//--------------------------------------------------------------
// Calculate master max surface speed [m/min]
//--------------------------------------------------------------
masterMaxSpeedMPM := groupMasterMaxSpeedRPM * (PI * upperMasterDiameter) / 1000.0;


//--------------------------------------------------------------
// Determine base speed source (auto/manual) + Recover bump
//--------------------------------------------------------------
IF groupSpeedAutoMan THEN
    baseCmdSpeedMPM := groupAutoSpeedMPM;
ELSE
    baseCmdSpeedMPM := groupManualSpeedMPM;
END_IF;

IF groupRecoverSpeedCmd THEN
    cmdSpeedMPM := baseCmdSpeedMPM + groupRecoverIncrement;
ELSE
    cmdSpeedMPM := baseCmdSpeedMPM;
END_IF;


//--------------------------------------------------------------
// Convert MPM → target RPM for the master
//--------------------------------------------------------------
targetRPM := _Scale(
    X    := cmdSpeedMPM,
    I_LO := 0.0,
    I_HI := masterMaxSpeedMPM,
    O_LO := 0.0,
    O_HI := groupMasterMaxSpeedRPM);


//--------------------------------------------------------------
// Ramp handling
//--------------------------------------------------------------
IF state = 5 OR state = 0 THEN
    // STOPPING — force ramp down to zero speed
    rampTargetRPM := 0.0;

ELSIF state = 10 THEN
    // FAULT — clear ramp immediately to ensure no residual motion
    rampTargetRPM := 0.0;
//    rampReset     := TRUE;

ELSE
    // Normal operation — ramp follows target speed
    rampTargetRPM := targetRPM;
//    rampReset     := FALSE;
END_IF;

// Detect when a new target speed change requires ramping
IF NOT (rampActive AND ABS(rampTargetRPM - baseMasterRefRPM) >= 0.05) OR NOT paperPresenceSensor THEN
   rampActive := TRUE; // Rising edge — ramp request detected
 
END_IF;


IF 	paperPresenceSensor THEN
	//slow	
	instFB_Gen_SRamp.A_UP := MAX(0.0, rampUpRate);
	instFB_Gen_SRamp.A_DN := -MAX(0.0, rampDownRate);

ELSE
	//fast
	instFB_Gen_SRamp.A_UP := MAX(0.0, rampUpRate2);
	instFB_Gen_SRamp.A_DN := -MAX(0.0, rampDownRate2);

END_IF


// Ramp function block execution
instFB_Gen_SRamp(
    X          := rampTargetRPM,
    VU_MAX     := 1000.0,
    VD_MAX     := -1000.0,
    LIMIT_HIGH := groupMasterMaxSpeedRPM,
    RST        := rampReset);


// If ramping, update the baseMasterRefRPM from ramp output
IF rampActive THEN
    baseMasterRefRPM := instFB_Gen_SRamp.Y;

    // Automatically reset ramp flag when the ramp output reaches the target
    IF ABS(instFB_Gen_SRamp.Y - rampTargetRPM) <= 0.05 THEN
        rampActive := FALSE; // Ramp complete
    END_IF;

ELSE
    // No ramping required — direct assignment
    baseMasterRefRPM := rampTargetRPM;
END_IF;


//--------------------------------------------------------------
// Operator offset (TUNE2 control)
//--------------------------------------------------------------
instTUNE2_GroupSpeedDiff(
    SET     := FALSE,
    SU      := groupSpeedDifInc,
    SD      := groupSpeedDifDec,
    RST     := FALSE,
    SS      := speedDifIncPerPulse,
    FS      := speedDifIncPerPulse,
    LIMIT_L := groupSpeedDifLimLow,
    LIMIT_H := groupSpeedDifLimHigh,
    Y       => groupSpeedOffset);

	
speedDif := groupSpeedOffset;
	
groupDeltaRatioAll  := 1.0 + (groupSpeedOffset * 0.01);
upperLowerBiasRatio := 1.0 + ((upperAndLowerSpeedOffset + upperAndLowerSpeedCalibration) * 0.01);


//--------------------------------------------------------------
// Apply offsets + calculate all drive RPM references
//--------------------------------------------------------------
upperMasterRefRPM := baseMasterRefRPM * groupDeltaRatioAll;
upperSlaveRefRPM := upperMasterRefRPM  * upperSlaveRatio;


lowerMasterRefRPM := upperMasterRefRPM * group1ToGroup2MasterRatio;
lowerSlaveRefRPM := lowerMasterRefRPM * lowerSlaveRatio;


//--------------------------------------------------------------
// Convert RPM → MPM (surface speeds)
//--------------------------------------------------------------
upperMasterRefMPM := upperMasterRefRPM * upperMasterDiameter * PI / 1000.0;
upperSlaveRefMPM := (upperSlaveRefRPM * upperSlaveDiameter * PI / 1000.0);


lowerMasterRefMPM := lowerMasterRefRPM * lowerMasterDiameter * PI / 1000.0;
lowerSlaveRefMPM := (lowerSlaveRefRPM * lowerSlaveDiameter * PI / 1000.0);


//--------------------------------------------------------------
// Suggest downstream handoff (group2 master surface speed)
//--------------------------------------------------------------
nextGroupSpeedRefMPM := upperMasterRefMPM;


//====================================================================
// ═══ PRIVATE METHOD — CALCULATE DIAMETER RATIOS ════════════════════
//====================================================================
METHOD PRIVATE _CalculateGearRatios
VAR_INPUT
END_VAR

//──────────────────────────────────────────────────────────────
// Gear Ratios — Group 1 (Reference: Group1 Master)
//──────────────────────────────────────────────────────────────
IF upperMasterDiameter > 0.0 THEN
    group1ToGroup2MasterRatio := upperMasterDiameter / lowerMasterDiameter;
    group1ToGroup1Slave1Ratio := upperMasterDiameter / upperSlaveDiameter;
ELSE
    group1ToGroup2MasterRatio := 0.0;
    group1ToGroup1Slave1Ratio := 0.0;
END_IF;

//──────────────────────────────────────────────────────────────
// Gear Ratios — Group 2 (Reference: Group2 Master)
//──────────────────────────────────────────────────────────────
IF lowerMasterDiameter > 0.0 THEN
    group2ToGroup2Slave1Ratio := lowerMasterDiameter / lowerSlaveDiameter;
ELSE
    group2ToGroup2Slave1Ratio := 0.0;
END_IF;
END_METHOD

METHOD PRIVATE _Scale : REAL
VAR_INPUT
    X    : REAL;
    I_LO : REAL;
    I_HI : REAL;
    O_LO : REAL;
    O_HI : REAL;
END_VAR
IF I_LO = I_HI THEN
	_Scale := O_LO;
ELSE
	_Scale := (O_HI - O_LO) / (I_HI - I_LO) * (LIMIT(I_LO, X, I_HI) - I_LO) + O_LO;
END_IF;
END_METHOD

END_FUNCTION_BLOCK

// ---- Function Blocks/PaperMachine/DriveControl/FB_WinderDriveControl_V1.TcPOU
FUNCTION_BLOCK FB_WinderDriveControl_V1
VAR_INPUT

    //==============================================================
    // GROUP INTERLOCKS & COMMANDS
    //==============================================================
    startGroup              : BOOL;  // EN: Start command (pulse) / PT: Comando de partida (pulso)
    stopGroup               : BOOL;  // EN: Stop command (maintained) / PT: Comando de parada (nível)
    groupReset              : BOOL;  // EN: Reset all group faults / PT: Reset geral de falhas do grupo
    
    disableGroup            : BOOL;  // EN: Disable the group operation / PT: Desabilitar operação do grupo

	enableTorqueControl		: BOOL;
	
	
	
    //==============================================================
    // SPEED OFFSET / MANUAL ADJUSTMENTS
    //==============================================================
    grouSpeedDifIncCmd      : BOOL;  // EN: Increase speed offset / PT: Aumenta o offset de velocidade
    grouSpeedDifDecCmd      : BOOL;  // EN: Decrease speed offset / PT: Reduz o offset de velocidade
    groupRecoverSpeedCmd    : BOOL;  // EN: Recover nominal speed while TRUE / PT: Recupera velocidade nominal enquanto TRUE

    // Pressure fine adjustments for rider roll
    pressureOperatorSideIncCmd : BOOL; // EN: Increase operator-side pressure / PT: Aumenta a pressão no lado do operador
    pressureOperatorSideDecCmd : BOOL; // EN: Decrease operator-side pressure / PT: Diminui a pressão no lado do operador

    pressureDriveSideIncCmd    : BOOL; // EN: Increase drive-side pressure / PT: Aumenta a pressão no lado motriz
    pressureDriveSideDecCmd    : BOOL; // EN: Decrease drive-side pressure / PT: Diminui a pressão no lado motriz

	riderRollWorkPositionCmd	: BOOL;
	riderRollReleasePositionCmd	: BOOL;
	
    //==============================================================
    // CORE LOCK (CHUCK LOCKING SYSTEM)
    //==============================================================
    coreLockAutoMan         : BOOL;  // EN: Core lock mode (0=Manual, 1=Auto) / PT: Modo do travamento do mandril (0=Manual, 1=Automático)
    coreLockCmd             : BOOL;  // EN: Lock core chucks / PT: Travar mandril (core chucks)
    coreUnlockCmd           : BOOL;  // EN: Unlock core chucks / PT: Destravar mandril

	//==============================================================
    // CORE LOCK (CHUCK LOCKING SYSTEM)
    //==============================================================
	coreAceleratorEngageCmd : BOOL;
	coreAceleratorDisengageCmd : BOOL;
	coreAceleratorMotorReady : BOOL;
	
    //==============================================================
    // CORE BRAKE CONTROL
    //==============================================================
    coreBrakeAutoMan        : BOOL;  // EN: Core brake mode (0=Manual, 1=Auto) / PT: Modo de freio do mandril (0=Manual, 1=Automático)
    coreBrakeEnableCmd      : BOOL;  // EN: Enable core brake / PT: Habilita o freio do mandril
    coreBrakeDisableCmd     : BOOL;  // EN: Disable core brake / PT: Desabilita o freio do mandril

    //==============================================================
    // DRIVE STATUS INPUTS — MAIN DRIVE
    //==============================================================
    masterReady             : BOOL;  // EN: Master drive ready (no trip) / PT: Drive mestre pronto (sem falha)

    //==============================================================
    // SPEED SETPOINTS & MODE SELECTION
    //==============================================================
    groupAutoSpeedMPM       : REAL;         // EN: Automatic mode line speed [m/min] / PT: Velocidade em modo automático [m/min]
    groupManualSpeedMPM     : REAL := 50.0; // EN: Manual mode line speed [m/min] / PT: Velocidade em modo manual [m/min]
    groupSpeedAutoMan       : BOOL;         // EN: Speed mode (0=Manual, 1=Auto) / PT: Modo de velocidade (0=Manual, 1=Automático)

    //==============================================================
    // SPEED & TORQUE FEEDBACKS — MASTER DRIVE
    //==============================================================
    masterSpeedFeedback     : REAL;  // EN: Actual speed feedback / PT: Velocidade real do drive
    masterTorqueFeedback    : REAL;  // EN: Actual torque feedback / PT: Torque real do drive

    //==============================================================
    // CORE POSITIONING ARM (PICK-UP ROLL)
    //==============================================================
    corePositioningArmFwdCmd      : BOOL;  // EN: Command to move arm forward / PT: Comando para avançar o braço posicionador
    corePositioningArmRevCmd      : BOOL;  // EN: Command to move arm backward / PT: Comando para recuar o braço posicionador

    corePositioningArmPosLimitFwd : BOOL;  // EN: Forward limit switch / PT: Fim de curso avançado
    corePositioningArmPosLimitRev : BOOL;  // EN: Reverse limit switch / PT: Fim de curso recuado

    corePositioningArmFault       : BOOL;  // EN: Positioning arm fault / PT: Falha no braço posicionador

    masterDiameter          : REAL := 263.878; // EN: Master drum diameter [mm] / PT: Diâmetro do rolo mestre [mm]

    //==============================================================
    // MACHINE CONFIGURATION STRUCT
    //==============================================================
    machineConfig : PaperMachine_TypeHmiConfig; // EN: Global HMI configuration / PT: Configuração global da HMI

END_VAR
VAR_OUTPUT

    //==============================================================
    // STATE & DIAGNOSTICS
    //==============================================================
    deviceState             : STRING; // EN: Current device state (text) / PT: Estado atual do grupo (texto)
    groupFault              : BOOL;   // EN: Group fault active / PT: Falha ativa no grupo
    statusCode              : INT;    // EN: 0=Idle, 1=Starting, 2=Running, 3=Fault / PT: 0=Parado, 1=Partindo, 2=Rodando, 3=Falha
	speedDif	: REAL;
    //==============================================================
    // DRIVE SPEED REFERENCES (RPM)
    //==============================================================
    masterSpeedSetpointRPM  : REAL;   // EN: Drive speed reference [RPM] / PT: Referência de velocidade do drive [RPM]

    //==============================================================
    // LINE SPEED & TORQUE REFERENCES
    //==============================================================
    nextGroupSpeedRefMPM    : REAL;   // EN: Speed reference for next group [m/min] / PT: Velocidade sugerida para o próximo grupo [m/min]

    //==============================================================
    // DRIVE ENABLE & RESET COMMANDS
    //==============================================================
    masterEnable            : BOOL;   // EN: Enable master drive / PT: Habilita o drive mestre

    //==============================================================
    // CORE POSITIONING ARM OUTPUTS
    //==============================================================
    corePositioningArmFwd   : BOOL;   // EN: Move arm forward / PT: Avançar braço posicionador
    corePositioningArmRev   : BOOL;   // EN: Move arm backward / PT: Recuar braço posicionador
	coreLockSolenoid		: BOOL;
	
	//==============================================================
    // CORE LOCK (CHUCK LOCKING SYSTEM)
    //==============================================================
	coreAceleratorEngageSolenoid : BOOL;
	coreAceleratorMotorStart 	: BOOL;	
	coreAceleratorMotorReset 	: BOOL;	
	
    //==============================================================
    // CORE BRAKE / LOCK OUTPUTS
    //==============================================================
    coreBrakeEnableSolenoid     : BOOL; // EN: Core brake solenoid 1 / PT: Solenóide do freio do mandril 1
    coreBrakeEnableSolenoid2    : BOOL; // EN: Core brake solenoid 2 / PT: Solenóide do freio do mandril 2

    //==============================================================
    // RIDER ROLL CONTROL (PRESSURE)
    //==============================================================
     riderRollSolenoid1               : BOOL; // EN: Rider roll engagement solenoid / PT: Solenóide de engate do rider roll
	 riderRollSolenoid2               : BOOL; // EN: Rider roll engagement solenoid / PT: Solenóide de engate do rider roll
 
   	pressureOperatorSideControllerOutput : REAL; // EN: Controller output (operator side) / PT: Saída do controlador (lado operador)
    pressureDriveSideControllerOutput    : REAL; // EN: Controller output (drive side) / PT: Saída do controlador (lado motriz)
   
	pressureSetpointOperatorSide : REAL; // EN: Controller output (operator side) / PT: Saída do controlador (lado operador)
    pressureSetpointDriveSide    : REAL; // EN: Controller output (drive side) / PT: Saída do controlador (lado motriz)

    //==============================================================
    // FEEDBACKS (LINE SPEED / TORQUE)
    //==============================================================
    upperMasterSpeedMPM      : REAL;  // EN: Line speed feedback [m/min] / PT: Velocidade de linha [m/min]
    upperMasterTorque        : REAL;  // EN: Master torque feedback / PT: Torque do mestre

    //==============================================================
    // HMI ALARMS STRUCT
    //==============================================================
    hmiAlarms                : PaperMachine_TypeHmiAlarms; // EN: Alarm structure / PT: Estrutura de alarmes

END_VAR

VAR
    //==============================================================
    // INTERNAL FUNCTION BLOCK INSTANCES
    //==============================================================
    instFB_GroupDriveControl_V1       : FB_GroupDriveControl_V1;  // EN: Core group logic / PT: Lógica principal do grupo
    instFB_GroupSpeedControl_V1       : FB_GroupSpeedControl_V1;  // EN: Speed regulation / PT: Controle de velocidade

    instFB_WinderSpeedControl       : FB_WinderSpeedControl;  // EN: Speed regulation / PT: Controle de velocidade

	
    instFB_GroupDisplayFilters_V1     : FB_GroupDisplayFilters_V1; // EN: Filters for HMI visualization / PT: Filtros de exibição para HMI


	instTONAdvanceTime: TON;
	rRiderRollWorkPositionCmd: BOOL;
	riderRollWorkPositionCmdOld: BOOL;
	rRiderRollReleasePositionCmd: BOOL;
	riderRollReleasePositionCmdOld: BOOL;
	instTONCoreAceleratorReturnTime: TON;
	
	operatorSideLastePressure : REAL;
	driveSideLastePressure : REAL;

	
	instTONCoreBrakeMaxTime: TON;
END_VAR

VAR PERSISTENT
	
	riderRollState	: INT;
    instTUNE2_PressureOperatorSide : TUNE2; // EN: PID for operator-side pressure / PT: PID da pressão lado operador
    instTUNE2_PressureDriveSide    : TUNE2; // EN: PID for drive-side pressure / PT: PID da pressão lado motriz

END_VAR

VAR_IN_OUT
	
	torqueSetpoint	: REAL;

END_VAR

// ─────────────────────────────────────────────────────────────────────────────
// MAIN CALL SEQUENCE
// ─────────────────────────────────────────────────────────────────────────────

_GroupControl();          // 1) State machine: edges, enables, stop modes

_alarmsDisplay();

_auxiliaryControls();
_CoreAceleratorControl();
_coreBrakeControl();
_coreLock();
_riderRollControl();

METHOD _alarmsDisplay
VAR_INPUT
END_VAR
END_METHOD

METHOD _auxiliaryControls
VAR_INPUT
END_VAR

//==============================================
// PICK-UP ROLL POSITIONER
//  - Uses: pickUpRollPosCmdFwd / pickUpRollPosCmdRev
//  - Safety: fault or limit reached → stop
//  - Safety (optional): if both cmds = TRUE, stop
//==============================================
IF NOT corePositioningArmFault THEN
    // Forward
    IF corePositioningArmFwdCmd
       AND NOT corePositioningArmRevCmd
       AND NOT corePositioningArmPosLimitFwd THEN
        // EN: run forward / PT: avança
        corePositioningArmFwd := TRUE;
    ELSE
        corePositioningArmFwd := FALSE;
    END_IF;

    // Reverse
    IF corePositioningArmRevCmd
       AND NOT corePositioningArmFwdCmd
       AND NOT corePositioningArmPosLimitRev THEN
        // EN: run reverse / PT: recua
        corePositioningArmRev := TRUE;
    ELSE
        corePositioningArmRev := FALSE;
    END_IF;
ELSE
    // EN: Fault → stop / PT: Falha → para
    corePositioningArmFwd := FALSE;
    corePositioningArmRev := FALSE;
END_IF;
END_METHOD

METHOD _CoreAceleratorControl
VAR_INPUT
END_VAR
(*


	//==============================================================
    // CORE LOCK (CHUCK LOCKING SYSTEM)
    //==============================================================
	coreAceleratorEngageSolenoid : BOOL;
	coreAceleratorMotorStart 	: BOOL;	
	coreAceleratorMotorReset 	: BOOL;	
	
		//==============================================================
    // CORE LOCK (CHUCK LOCKING SYSTEM)
    //==============================================================
	coreAceleratorEngageCmd : BOOL;
	coreAceleratorDisengageCmd : BOOL;
	coreAceleratorMotorReady : BOOL;

*)


//IF NOT coreAceleratorMotorReady THEN
	
	IF coreAceleratorEngageCmd AND NOT coreAceleratorDisengageCmd THEN
		
		instTONCoreAceleratorReturnTime.IN := TRUE;
		coreAceleratorEngageSolenoid := TRUE;
		coreAceleratorMotorStart := TRUE;
	
	END_IF
	
	
	
	IF (coreAceleratorDisengageCmd AND NOT coreAceleratorEngageCmd) OR instTONCoreAceleratorReturnTime.Q THEN
		
		instTONCoreAceleratorReturnTime.IN := FALSE;
		coreAceleratorEngageSolenoid := FALSE;	
		coreAceleratorMotorStart := FALSE;
		
	
	END_IF
	
//END_IF



instTONCoreAceleratorReturnTime(PT := T#30S);
END_METHOD

METHOD _coreBrakeControl
 

IF coreBrakeEnableCmd AND NOT coreBrakeDisableCmd THEN
	
	coreBrakeEnableSolenoid := TRUE;
	instTONCoreBrakeMaxTime.IN := TRUE;	
	
END_IF

IF (coreBrakeDisableCmd AND NOT coreBrakeEnableCmd) OR instTONCoreBrakeMaxTime.Q  THEN
	
	coreBrakeEnableSolenoid := FALSE;
	instTONCoreBrakeMaxTime.IN := FALSE;	
	

END_IF


instTONCoreBrakeMaxTime(PT := T#10S);
END_METHOD

METHOD _coreLock

IF corePositioningArmPosLimitFwd OR corePositioningArmPosLimitRev THEN
	
	IF coreLockCmd AND NOT coreUnlockCmd THEN
		
		coreLockSolenoid := TRUE;
	
	END_IF
	
	IF coreUnlockCmd AND NOT coreLockCmd THEN
		
		coreLockSolenoid := FALSE;

	END_IF

END_IF
END_METHOD

METHOD _GroupControl
VAR_INPUT
END_VAR
(*
FUNCTION_BLOCK FB_DryingSectionDriveControl_V3
VAR_INPUT

    //==============================================================
    // GROUP INTERLOCKS & COMMANDS
    //==============================================================
    startGroup              : BOOL;  // EN: Start command (pulse) / PT: Comando de partida (pulso)
    stopGroup               : BOOL;  // EN: Stop command (level) / PT: Comando de parada (nível)
    groupReset              : BOOL;  // EN: Reset group faults / PT: Reset de falhas do grupo

    //==============================================================
    // SPEED OFFSET / MANUAL ADJUSTMENTS
    //==============================================================
    grouSpeedDifIncCmd      : BOOL;  // EN: Lamp or indication – speed offset increasing / PT: Lâmpada ou indicação – offset de velocidade aumentando
    grouSpeedDifDecCmd      : BOOL;  // EN: Lamp or indication – speed offset decreasing / PT: Lâmpada ou indicação – offset de velocidade reduzindo
    groupRecoverSpeedCmd    : BOOL;  // EN: Recover nominal speed while TRUE / PT: Recuperar velocidade nominal enquanto TRUE

    //==============================================================
    // DRIVE STATUS INPUTS — UPPER GROUP
    //==============================================================
    upperMasterReady        : BOOL;  // EN: Upper master ready (no trip) / PT: Mestre superior pronto (sem falha)
    upperSlave1Ready        : BOOL;  // EN: Upper slave 1 ready / PT: Escravo 1 superior pronto

    //==============================================================
    // DRIVE STATUS INPUTS — LOWER GROUP
    //==============================================================
    lowerMasterReady        : BOOL;  // EN: Lower master ready (no trip) / PT: Mestre inferior pronto (sem falha)
    lowerSlave1Ready        : BOOL;  // EN: Lower slave 1 ready / PT: Escravo 1 inferior pronto

    //==============================================================
    // SPEED SETPOINTS & MODE SELECTION
    //==============================================================
    groupAutoSpeedMPM       : REAL;        // EN: Automatic mode speed [m/min] / PT: Velocidade em modo automático [m/min]
    groupManualSpeedMPM     : REAL := 50.0;// EN: Manual mode speed [m/min] / PT: Velocidade em modo manual [m/min]
    groupSpeedAutoMan       : BOOL;        // EN: Speed mode (0=Manual, 1=Auto) / PT: Modo de velocidade (0=Manual, 1=Automático)

    //==============================================================
    // SPEED & TORQUE FEEDBACKS — UPPER GROUP
    //==============================================================
    upperMasterSpeedFeedback    : REAL;  // [m/min or %]
    upperMasterTorqueFeedback   : REAL;  // [% or Nm]
    upperSlave1SpeedFeedback    : REAL;
    upperSlave1TorqueFeedback   : REAL;

    //==============================================================
    // SPEED & TORQUE FEEDBACKS — LOWER GROUP
    //==============================================================
    lowerMasterSpeedFeedback    : REAL;
    lowerMasterTorqueFeedback   : REAL;
    lowerSlave1SpeedFeedback    : REAL;
    lowerSlave1TorqueFeedback   : REAL;

    //==============================================================
    // COOLING MOTOR FAULT INPUTS
    //==============================================================
    upperMasterCoolingMotorFault : BOOL;  // EN: Upper master cooling motor fault / PT: Falha no motor de ventilação do mestre superior
    upperSlave1CoolingMotorFault : BOOL;  // EN: Upper slave 1 cooling motor fault / PT: Falha no motor de ventilação do escravo 1 superior
    lowerMasterCoolingMotorFault : BOOL;  // EN: Lower master cooling motor fault / PT: Falha no motor de ventilação do mestre inferior
    lowerSlave1CoolingMotorFault : BOOL;  // EN: Lower slave 1 cooling motor fault / PT: Falha no motor de ventilação do escravo 1 inferior

    //==============================================================
    // FABRIC / WIRE STRETCHER ACTUATORS
    //==============================================================
    upperDryingSectionFabricStretchCmd     : BOOL;  // EN: Command to stretch upper fabric / PT: Comando para esticar a tela superior
    upperDryingSectionFabricUnstretchCmd   : BOOL;  // EN: Command to loosen upper fabric / PT: Comando para afrouxar a tela superior
    lowerDryingSectionFabricStretchCmd     : BOOL;  // EN: Command to stretch lower fabric / PT: Comando para esticar a tela inferior
    lowerDryingSectionFabricUnstretchCmd   : BOOL;  // EN: Command to loosen lower fabric / PT: Comando para afrouxar a tela inferior
    upperDryingSectionFabricStretcherMotorFault : BOOL;  // EN: Upper stretcher motor fault / PT: Falha no motor de estiramento superior
    lowerDryingSectionFabricStretcherMotorFault : BOOL;  // EN: Lower stretcher motor fault / PT: Falha no motor de estiramento inferior

    //==============================================================
    // FABRIC / WIRE OVERRUN SENSORS
    //==============================================================
    upperDryingSectionFabricOverrunOperatorSideSensor : BOOL; // EN: Upper fabric overrun sensor (operator side) / PT: Sensor de sobrecurso da tela superior (lado operador)
    upperDryingSectionFabricOverrunDriveSideSensor    : BOOL; // EN: Upper fabric overrun sensor (drive side) / PT: Sensor de sobrecurso da tela superior (lado acionamento)
    lowerDryingSectionFabricOverrunOperatorSideSensor : BOOL; // EN: Lower fabric overrun sensor (operator side) / PT: Sensor de sobrecurso da tela inferior (lado operador)
    lowerDryingSectionFabricOverrunDriveSideSensor    : BOOL; // EN: Lower fabric overrun sensor (drive side) / PT: Sensor de sobrecurso da tela inferior (lado acionamento)

    //==============================================================
    // PICK-UP ROLL POSITIONER
    //==============================================================
    pickUpRollPosCmdFwd       : BOOL;  // EN: Command forward / PT: Avanço do rolo pick-up
    pickUpRollPosCmdRev       : BOOL;  // EN: Command reverse / PT: Recuo do rolo pick-up
    pickUpRollPosLimitFwd     : BOOL;  // EN: Forward limit switch / PT: Fim de curso frontal
    pickUpRollPosLimitRev     : BOOL;  // EN: Reverse limit switch / PT: Fim de curso traseiro
    pickUpRollPosFault        : BOOL;  // EN: Positioner fault / PT: Falha no posicionador

    //==============================================================
    // SCRAPER OSCILLATORS
    //==============================================================
    babyDryerScraperOscCmd     : BOOL;  // EN: Command to start Baby Dryer scraper oscillator / PT: Comando para iniciar oscilador do Baby Dryer
    babyDryerScraperOscFault   : BOOL;  // EN: Baby Dryer oscillator fault / PT: Falha no oscilador do Baby Dryer
    babyDryerScraperOscRunning : BOOL;  // EN: Baby Dryer oscillator running / PT: Oscilador do Baby Dryer em operação

    upperGroupScraperOscCmd     : BOOL;  // EN: Upper group scraper oscillator command / PT: Comando de oscilação da raspa do grupo superior
    upperGroupScraperOscFault   : BOOL;  // EN: Upper group oscillator fault / PT: Falha no oscilador do grupo superior
    upperGroupScraperOscRunning : BOOL;  // EN: Upper group oscillator running / PT: Oscilador do grupo superior em operação

    lowerGroupScraperOscCmd     : BOOL;  // EN: Lower group scraper oscillator command / PT: Comando de oscilação da raspa do grupo inferior
    lowerGroupScraperOscFault   : BOOL;  // EN: Lower group oscillator fault / PT: Falha no oscilador do grupo inferior
    lowerGroupScraperOscRunning : BOOL;  // EN: Lower group oscillator running / PT: Oscilador do grupo inferior em operação

    //==============================================================
    // STEAM PRESSURE CONTROL (PID)
    //==============================================================
    steamPressureAutoMan        : BOOL;  // EN: Steam pressure mode (0=Manual, 1=Auto) / PT: Modo de pressão do vapor (0=Manual, 1=Automático)
    steamPressureAutoSetpoint   : REAL;  // EN: Auto mode setpoint [bar] / PT: Setpoint em modo automático [bar]
    steamPressureManualSetpoint : REAL;  // EN: Manual mode setpoint [bar] / PT: Setpoint em modo manual [bar]
    steamPressureFeedback       : REAL;  // EN: Steam pressure feedback [bar] / PT: Retorno de pressão do vapor [bar]
    steamPressureKp             : REAL := 1.0;  // EN: PID proportional gain / PT: Ganho proporcional do PID
    steamPressureTn             : REAL := 8.0;  // EN: PID integral time [s] / PT: Tempo integral do PID [s]
    steamPressureTv             : REAL := 0.0;  // EN: PID derivative time [s] / PT: Tempo derivativo do PID [s]

    //==============================================================
    // MACHINE CONFIGURATION STRUCT
    //==============================================================
    machineConfig               : PaperMachine_TypeHmiConfig; // EN: HMI configuration structure / PT: Estrutura de configuração da HMI

END_VAR
	winderDiameter	: REAL := 800.9;
	winderMotorRPM	: REAL := 212.5; //Motor RPM  / Rel. Mecanicia (1700 / 8)
	


VAR_OUTPUT

    //==============================================================
    // STATE & DIAGNOSTICS
    //==============================================================
    deviceState                 : STRING;  // EN: Current readable device state / PT: Estado textual atual do grupo
    groupFault                  : BOOL;    // EN: Group fault active / PT: Falha ativa no grupo
    statusCode                  : INT;     // EN: 0=Idle, 1=Starting, 2=Running, 3=Fault / PT: 0=Parado, 1=Partindo, 2=Rodando, 3=Falha

    //==============================================================
    // DRIVE SPEED REFERENCES (RPM)
    //==============================================================
    upperMasterSpeedSetpointRPM : REAL;
    upperSlaveSpeedSetpointRPM  : REAL;
    lowerMasterSpeedSetpointRPM : REAL;
    lowerSlaveSpeedSetpointRPM  : REAL;


    //==============================================================
    // LINE SPEED & TORQUE REFERENCES
    //==============================================================
    nextGroupSpeedRefMPM        : REAL;  // EN: Suggested next group speed [m/min] / PT: Velocidade sugerida para o próximo grupo [m/min]

    upperSlave1TorqueRefPct     : REAL;
    upperSlave2TorqueRefPct     : REAL;
    lowerSlave1TorqueRefPct     : REAL;
    lowerSlave2TorqueRefPct     : REAL;

    //==============================================================
    // DRIVE ENABLE & RESET COMMANDS
    //==============================================================
    upperMasterEnable           : BOOL;
    upperSlave1Enable           : BOOL;
    upperMasterReset            : BOOL;
    upperSlave1Reset            : BOOL;

    lowerMasterEnable           : BOOL;
    lowerSlave1Enable           : BOOL;
    lowerMasterReset            : BOOL;
    lowerSlave1Reset            : BOOL;

    //==============================================================
    // FABRIC / WIRE STRETCHERS
    //==============================================================
    upperDryingSectionFabricStretch   : BOOL;
    upperDryingSectionFabricUnstretch : BOOL;
    lowerDryingSectionFabricStretch   : BOOL;
    lowerDryingSectionFabricUnstretch : BOOL;

    //==============================================================
    // PICK-UP ROLL POSITIONER OUTPUTS
    //==============================================================
    pickUpRollPosRunFwd          : BOOL;
    pickUpRollPosRunRev          : BOOL;

    //==============================================================
    // SCRAPER OSCILLATORS OUTPUTS
    //==============================================================
    babyDryerScraperOscRun       : BOOL;
    upperGroupScraperOscRun      : BOOL;
    lowerGroupScraperOscRun      : BOOL;

    //==============================================================
    // STEAM PRESSURE PID OUTPUT
    //==============================================================
    steamPressureControllerOutput : REAL;

    //==============================================================
    //FEEDBACKS (MPM / RPM / TOQUE)
    //==============================================================
    upperMasterSpeedMPM          : REAL;
    upperSlave1SpeedMPM          : REAL;
    lowerMasterSpeedMPM          : REAL;
    lowerSlave1SpeedMPM          : REAL;

    upperMasterSpeedRPM          : REAL;
    upperSlave1SpeedRPM          : REAL;
    lowerMasterSpeedRPM          : REAL;
    lowerSlave1SpeedRPM          : REAL;
	
    upperMasterTorque          	: REAL;
    upperSlave1Torqu          	: REAL;
    lowerMasterTorque          	: REAL;
    lowerSlave1Torque          	: REAL;

    //==============================================================
    // HMI ALARMS STRUCT
    //==============================================================
    hmiAlarms                    : PaperMachine_TypeHmiAlarms;

END_VAR



VAR
    //==============================================================
    // INTERNAL FUNCTION BLOCK INSTANCES
    //==============================================================
    instFB_GroupDriveControl_V1       : FB_GroupDriveControl_V1;
    instFB_GroupSpeedControl_V1       : FB_GroupSpeedControl_V1;
    instFB_GroupDisplayFilters_V1     : FB_GroupDisplayFilters_V1;
    instFB_GroupTorqueTrimControl_V1  : FB_GroupTorqueTrimControl_V1;
    instCTRL_PID_TemperatureController: CTRL_PID;

END_VAR



VAR PERSISTENT
    //==============================================================
    // TUNING PARAMETERS (PERSISTENT)
    //==============================================================
    instTUNE2_GroupSpeedDiference     : TUNE2; // EN: Manual tuning helper for group speed difference / PT: Auxiliar de ajuste manual da diferença de velocidade do grupo
END_VAR

	masterDiameter := 795	
*)
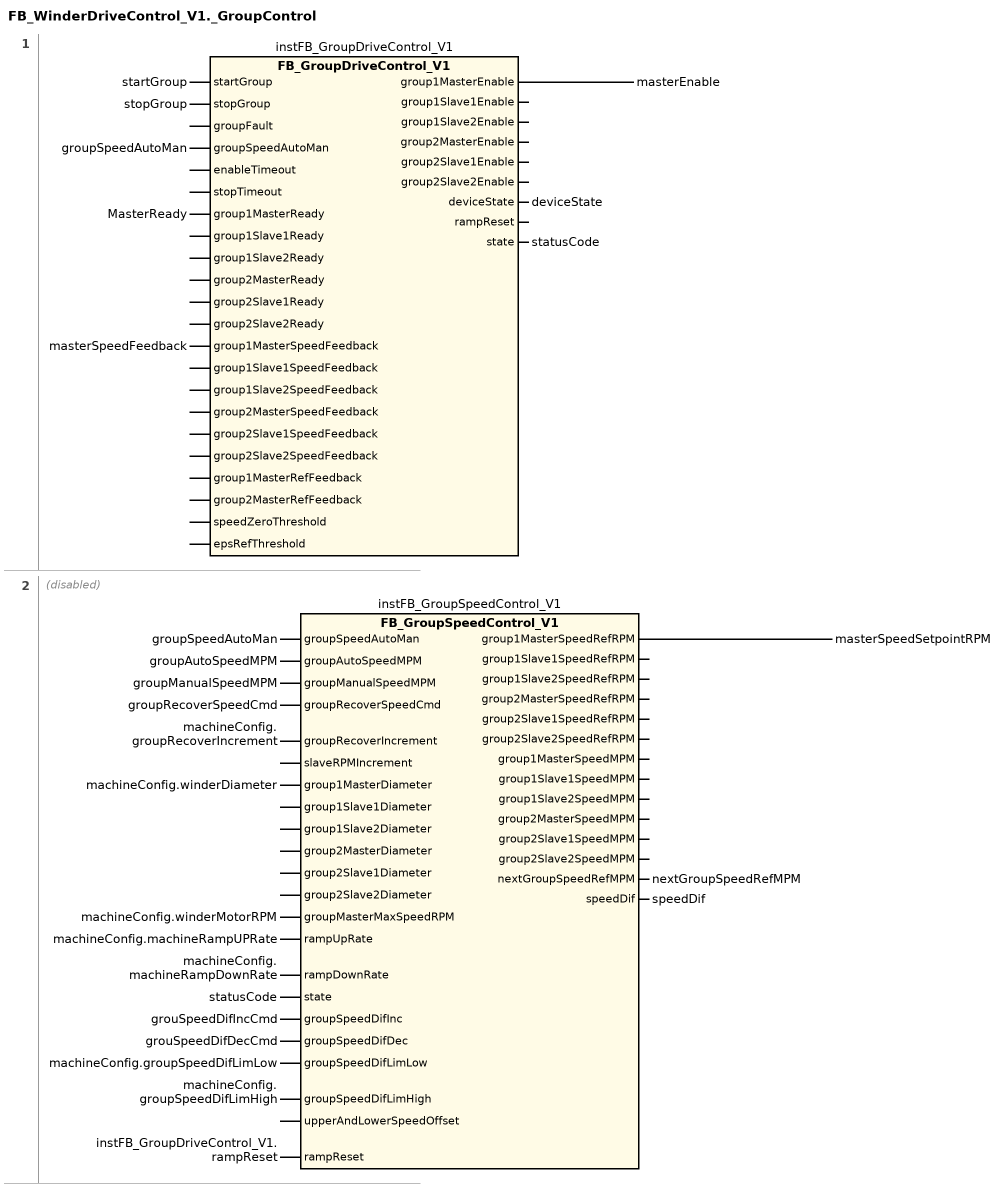
// NETWORK 1
instFB_GroupDriveControl_V1(
    startGroup := startGroup,
    stopGroup := stopGroup,
    groupSpeedAutoMan := groupSpeedAutoMan,
    group1MasterReady := MasterReady,
    group1MasterSpeedFeedback := masterSpeedFeedback,
    deviceState => deviceState,
    state => statusCode); // FB_GroupDriveControl_V1
masterEnable := instFB_GroupDriveControl_V1.group1MasterEnable;

// NETWORK 2 (disabled)
// instFB_GroupSpeedControl_V1(
//     groupSpeedAutoMan := groupSpeedAutoMan,
//     groupAutoSpeedMPM := groupAutoSpeedMPM,
//     groupManualSpeedMPM := groupManualSpeedMPM,
//     groupRecoverSpeedCmd := groupRecoverSpeedCmd,
//     groupRecoverIncrement := machineConfig.groupRecoverIncrement,
//     group1MasterDiameter := machineConfig.winderDiameter,
//     groupMasterMaxSpeedRPM := machineConfig.winderMotorRPM,
//     rampUpRate := machineConfig.machineRampUPRate,
//     rampDownRate := machineConfig.machineRampDownRate,
//     state := statusCode,
//     groupSpeedDifInc := grouSpeedDifIncCmd,
//     groupSpeedDifDec := grouSpeedDifDecCmd,
//     groupSpeedDifLimLow := machineConfig.groupSpeedDifLimLow,
//     groupSpeedDifLimHigh := machineConfig.groupSpeedDifLimHigh,
//     rampReset := instFB_GroupDriveControl_V1.rampReset,
//     nextGroupSpeedRefMPM => nextGroupSpeedRefMPM,
//     speedDif => speedDif); // FB_GroupSpeedControl_V1
// masterSpeedSetpointRPM := instFB_GroupSpeedControl_V1.group1MasterSpeedRefRPM;

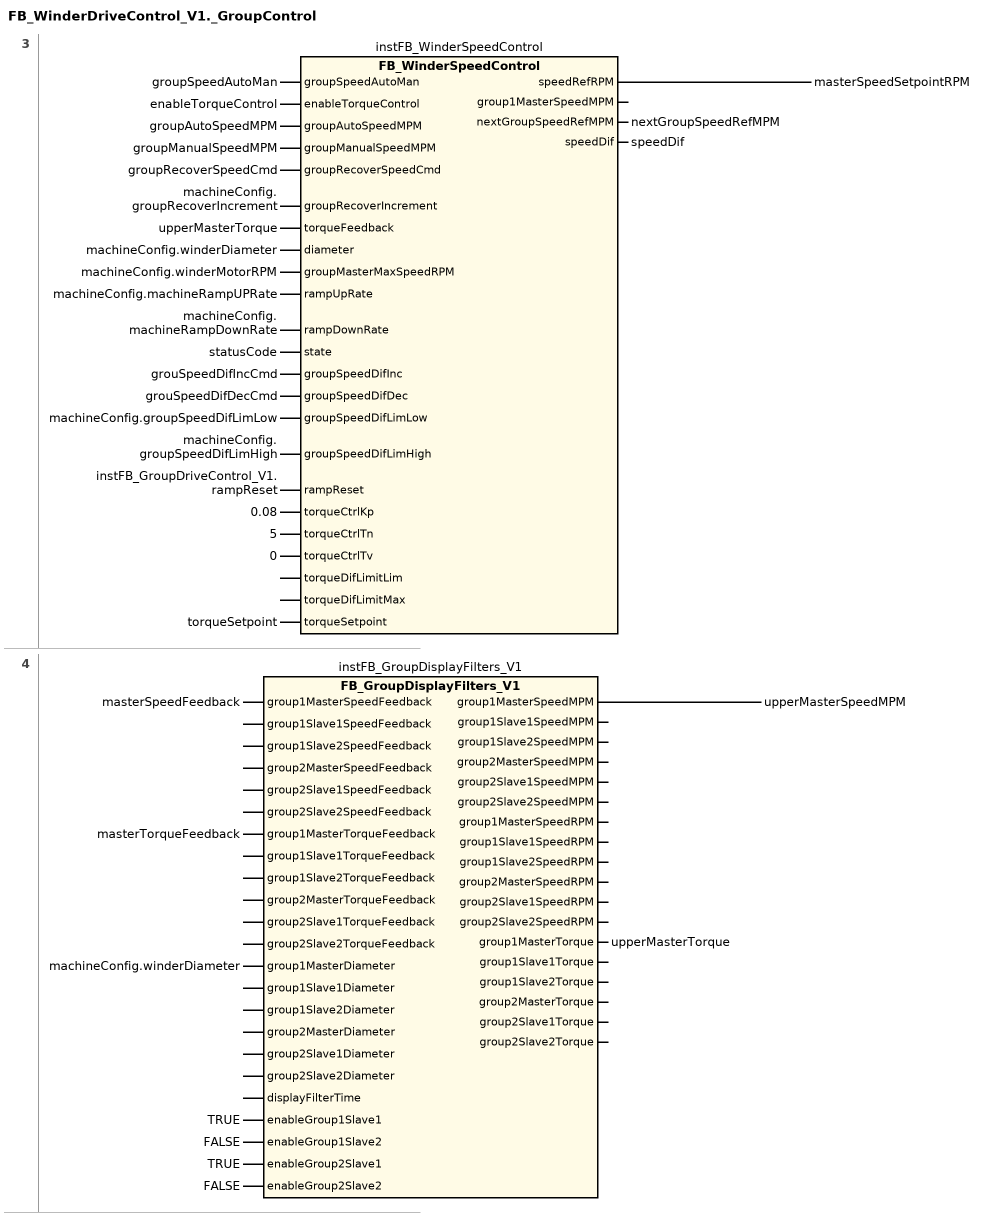
// NETWORK 3
instFB_WinderSpeedControl(
    groupSpeedAutoMan := groupSpeedAutoMan,
    enableTorqueControl := enableTorqueControl,
    groupAutoSpeedMPM := groupAutoSpeedMPM,
    groupManualSpeedMPM := groupManualSpeedMPM,
    groupRecoverSpeedCmd := groupRecoverSpeedCmd,
    groupRecoverIncrement := machineConfig.groupRecoverIncrement,
    torqueFeedback := upperMasterTorque,
    diameter := machineConfig.winderDiameter,
    groupMasterMaxSpeedRPM := machineConfig.winderMotorRPM,
    rampUpRate := machineConfig.machineRampUPRate,
    rampDownRate := machineConfig.machineRampDownRate,
    state := statusCode,
    groupSpeedDifInc := grouSpeedDifIncCmd,
    groupSpeedDifDec := grouSpeedDifDecCmd,
    groupSpeedDifLimLow := machineConfig.groupSpeedDifLimLow,
    groupSpeedDifLimHigh := machineConfig.groupSpeedDifLimHigh,
    rampReset := instFB_GroupDriveControl_V1.rampReset,
    torqueCtrlKp := 0.08,
    torqueCtrlTn := 5,
    torqueCtrlTv := 0,
    torqueSetpoint := torqueSetpoint,
    nextGroupSpeedRefMPM => nextGroupSpeedRefMPM,
    speedDif => speedDif); // FB_WinderSpeedControl
masterSpeedSetpointRPM := instFB_WinderSpeedControl.speedRefRPM;

// NETWORK 4
instFB_GroupDisplayFilters_V1(
    group1MasterSpeedFeedback := masterSpeedFeedback,
    group1MasterTorqueFeedback := masterTorqueFeedback,
    group1MasterDiameter := machineConfig.winderDiameter,
    enableGroup1Slave1 := TRUE,
    enableGroup1Slave2 := FALSE,
    enableGroup2Slave1 := TRUE,
    enableGroup2Slave2 := FALSE,
    group1MasterTorque => upperMasterTorque); // FB_GroupDisplayFilters_V1
upperMasterSpeedMPM := instFB_GroupDisplayFilters_V1.group1MasterSpeedMPM;
END_METHOD

METHOD _riderRollControl


(*
	operatorSideLastePressure : REAL;
	driveSideLastePressure : REAL;
	
	riderRollWorkPositionCmd	: BOOL;
	riderRollReleasePositionCmd	: BOOL;


*)


rRiderRollWorkPositionCmd := riderRollWorkPositionCmd AND NOT riderRollWorkPositionCmdOld;

rRiderRollReleasePositionCmd := riderRollReleasePositionCmd AND NOT riderRollReleasePositionCmdOld;
 

	
IF rRiderRollWorkPositionCmd THEN
	
	riderRollState := 2;
	
END_IF


IF rRiderRollReleasePositionCmd THEN
	
	riderRollState := 1;

END_IF

riderRollWorkPositionCmdOld := riderRollWorkPositionCmd;
riderRollReleasePositionCmdOld := riderRollReleasePositionCmd;

//==============================================================
// State machine (Rider Roll)
//==============================================================
CASE riderRollState OF

//------------------------------------------------------------------
// 0: IDLE
//------------------------------------------------------------------
0:

	instTONAdvanceTime.IN := FALSE;


//------------------------------------------------------------------
// 1: RELEASE POSITION - PRESSURE TO MIN VALUE
//------------------------------------------------------------------
1:

	//Save the last setpoint
	operatorSideLastePressure := instTUNE2_PressureOperatorSide.Y;
	driveSideLastePressure := instTUNE2_PressureDriveSide.Y;

    instTUNE2_PressureOperatorSide.SET_val := 0.0;  // Max pressure
    instTUNE2_PressureOperatorSide.SET := TRUE;
	instTUNE2_PressureOperatorSide();
	
    instTUNE2_PressureDriveSide.SET_val := 0.0;  // Max pressure
    instTUNE2_PressureDriveSide.SET := TRUE;
	instTUNE2_PressureDriveSide();

    // Command solenoid to release position
    riderRollSolenoid1 := TRUE;
    riderRollSolenoid2 := TRUE;
	
	
	//Wait for command
	riderRollState := 0;




//------------------------------------------------------------------
// 2: FAST ADVANCE - PRESSURE TO MAX VALUE
//------------------------------------------------------------------
2:
    // Initial pressure for fast approach

	
    instTUNE2_PressureOperatorSide.SET_val := 9.0;  // Max pressure
    instTUNE2_PressureOperatorSide.SET := TRUE;
	instTUNE2_PressureOperatorSide();
	
    instTUNE2_PressureDriveSide.SET_val := 9.0;  // Max pressure
    instTUNE2_PressureDriveSide.SET := TRUE;
	instTUNE2_PressureDriveSide();
	
    // Advance solenoid
    riderRollSolenoid1 := FALSE;
    riderRollSolenoid2 := FALSE;

    instTONAdvanceTime.IN := TRUE;

    // When timer finishes, go to work mode
    IF instTONAdvanceTime.Q THEN
	
        instTONAdvanceTime.IN := FALSE;
        riderRollState := 3;  // Enter WORK POSITION
		
    END_IF



//------------------------------------------------------------------
// 3: GO TO WORK POSITION - PRESSURE START VALUE
//------------------------------------------------------------------
3:

	instTUNE2_PressureOperatorSide.SET_val := 0.8;
	instTUNE2_PressureOperatorSide.SET := TRUE;
	instTUNE2_PressureOperatorSide();
		
	instTUNE2_PressureDriveSide.SET_val := 0.8;
	instTUNE2_PressureDriveSide.SET := TRUE;
	instTUNE2_PressureDriveSide();

		
    // Solenoid keeps rider roll engaged
    riderRollSolenoid1 := FALSE;
    riderRollSolenoid2 := FALSE;

	//Wait for command
	riderRollState := 0;


END_CASE



//==============================================================
// Timers execution
//==============================================================
instTONAdvanceTime(PT := machineConfig.winderRiderRollAdvTime);


//==============================================================
// Operator side pressure PID (offset tuning)
//==============================================================
instTUNE2_PressureOperatorSide(
    SU      := pressureOperatorSideIncCmd,
    SD      := pressureOperatorSideDecCmd,
	SET 	:= FALSE,
    SS      := 0.1,
    FS      := 1.0,
    LIMIT_L := 0.0,
    LIMIT_H := 9.0,
    Y       => pressureOperatorSideControllerOutput);


//==============================================================
// Drive side pressure PID
//==============================================================
instTUNE2_PressureDriveSide(
    SU      := pressureDriveSideIncCmd,
    SD      := pressureDriveSideDecCmd,
	SET 	:= FALSE,
    SS      := 0.1,
    FS      := 1.0,
    LIMIT_L := 0.0,
    LIMIT_H := 9.0,
    Y       => pressureDriveSideControllerOutput);
	
	
	   
	pressureSetpointOperatorSide := pressureOperatorSideControllerOutput;
    pressureSetpointDriveSide    := pressureDriveSideControllerOutput;
END_METHOD

END_FUNCTION_BLOCK

// ---- Function Blocks/PaperMachine/FB_WinderSpeedControl.TcPOU
FUNCTION_BLOCK FB_WinderSpeedControl
VAR_INPUT
    //==============================================================
    // ─────────────── MODE SELECTION / REFERENCES ───────────────
    //==============================================================
    groupSpeedAutoMan          : BOOL;  // TRUE = Auto, FALSE = Manual
    enableTorqueControl          : BOOL;  // TRUE = Auto, FALSE = Manual

    groupAutoSpeedMPM          : REAL;  // Auto speed reference [m/min]
    groupManualSpeedMPM        : REAL;  // Manual speed reference [m/min]
    groupRecoverSpeedCmd       : BOOL;  // Recover (temporary speed bump)
    groupRecoverIncrement      : REAL;  // Recover increment [m/min]

	
	torqueFeedback				: REAL;
    //==============================================================
    // ─────────────── DIAMETERS (mm) ───────────────
    //==============================================================
    diameter       : REAL;  // Diameter of group 1 master

    //==============================================================
    // ─────────────── CONFIGURATION / LIMITS ───────────────
    //==============================================================
    groupMasterMaxSpeedRPM     : REAL;  		// Max allowed master RPM
    rampUpRate					: REAL := 0.1;  // Ramp acceleration [RPM/s]
    rampDownRate				: REAL := 0.1;  // Ramp acceleration [RPM/s]
	
    state                      : INT;   // Machine state (5 = STOPPING)

    groupSpeedDifInc           : BOOL;  // Increment group speed offset
    groupSpeedDifDec           : BOOL;  // Decrement group speed offset
    groupSpeedDifLimLow        : REAL;  // Min offset [%]
    groupSpeedDifLimHigh       : REAL;  // Max offset [%]

    rampReset                  : BOOL;  // Reset ramp command
	
	
    torqueCtrlKp                   : REAL := 0.50;
    torqueCtrlTn                   : REAL := 5.0;
    torqueCtrlTv                   : REAL := 0.0;
	torqueDifLimitLim				: REAL := -3.0;
	torqueDifLimitMax				: REAL := 3.0;	
	
	
	
	
END_VAR


VAR_OUTPUT
    //==============================================================
    // ─────────────── FINAL DRIVE SPEEDS (RPM) ───────────────
    //==============================================================
    speedRefRPM    : REAL;


    //==============================================================
    // ─────────────── SURFACE SPEEDS (MPM) ───────────────
    //==============================================================
    group1MasterSpeedMPM       : REAL;


    //==============================================================
    // ─────────────── HANDOFF TO NEXT GROUP ───────────────
    //==============================================================
    nextGroupSpeedRefMPM       : REAL;
	speedDif					: REAL;
	
END_VAR


VAR
    //==============================================================
    // ─────────────── INTERNAL CALCULATION VARIABLES ───────────────
    //==============================================================
    masterMaxSpeedMPM          : REAL;
    baseCmdSpeedMPM            : REAL;
    cmdSpeedMPM                : REAL;
    targetRPM                  : REAL;
    rampTargetRPM              : REAL;
    baseMasterRefRPM           : REAL;
    groupSpeedOffset           : REAL;
    groupDeltaRatioAll         : REAL;
    upperLowerBiasRatio        : REAL;
    useRamp                    : BOOL;
    epsDiameter                : REAL := 0.001;

    // Gear ratios (set externally or calculated elsewhere)
    group1ToGroup1Slave1Ratio  : REAL := 1.0;
    group1ToGroup1Slave2Ratio  : REAL := 1.0;
    group1ToGroup2MasterRatio  : REAL := 1.0;
    group2ToGroup2Slave1Ratio  : REAL := 1.0;
    group2ToGroup2Slave2Ratio  : REAL := 1.0;

    // Function blocks
    instFB_Gen_SRamp           : FB_Gen_SRamp;
    speedOffsetPID   : REAL;  // Bias [%] between group1 and group2
 	instCTRL_PID_Group1TorqueTrim : CTRL_PID;
	rampActive: BOOL;
	enableTorqueControlOld: BOOL;
END_VAR

VAR_IN_OUT
	
	torqueSetpoint	: REAL;

END_VAR
VAR PERSISTENT
	
    instTUNE2_GroupSpeedDiff   : TUNE2;

END_VAR

//==============================================================
// IMPLEMENTATION
//==============================================================

//====================================================================
// ═══ CALL METHOD TO CALCULATE DIAMETER RATIOS ═════════════════════
//====================================================================
_CalculateGearRatios();

//--------------------------------------------------------------
// Calculate master max surface speed [m/min]
//--------------------------------------------------------------
masterMaxSpeedMPM := groupMasterMaxSpeedRPM * (PI * diameter) / 1000.0;


//--------------------------------------------------------------
// Determine base speed source (auto/manual) + Recover bump
//--------------------------------------------------------------
IF groupSpeedAutoMan THEN
    baseCmdSpeedMPM := groupAutoSpeedMPM;
ELSE
    baseCmdSpeedMPM := groupManualSpeedMPM;
END_IF;

IF groupRecoverSpeedCmd THEN
    cmdSpeedMPM := baseCmdSpeedMPM + groupRecoverIncrement;
ELSE
    cmdSpeedMPM := baseCmdSpeedMPM;
END_IF;


//--------------------------------------------------------------
// Convert MPM → target RPM for the master
//--------------------------------------------------------------
targetRPM := _Scale(
    X    := cmdSpeedMPM,
    I_LO := 0.0,
    I_HI := masterMaxSpeedMPM,
    O_LO := 0.0,
    O_HI := groupMasterMaxSpeedRPM);


//--------------------------------------------------------------
// Ramp handling
//--------------------------------------------------------------
IF state = 5 OR state = 0 THEN
    // STOPPING — force ramp down to zero speed
    rampTargetRPM := 0.0;

ELSIF state = 10 THEN
    // FAULT — clear ramp immediately to ensure no residual motion
    rampTargetRPM := 0.0;
//    rampReset     := TRUE;

ELSE
    // Normal operation — ramp follows target speed
    rampTargetRPM := targetRPM;
//    rampReset     := FALSE;
END_IF;

// Detect when a new target speed change requires ramping
IF NOT rampActive AND ABS(rampTargetRPM - baseMasterRefRPM) >= 1.0 THEN
   rampActive := TRUE; // Rising edge — ramp request detected
 
END_IF;

// Ramp function block execution
instFB_Gen_SRamp(
    X          := rampTargetRPM,
    A_UP       := MAX(0.0, rampUpRate),
    A_DN       := -MAX(0.0, rampDownRate),
    VU_MAX     := 1000.0,
    VD_MAX     := -1000.0,
    LIMIT_HIGH := groupMasterMaxSpeedRPM,
    RST        := rampReset);

// If ramping, update the baseMasterRefRPM from ramp output
IF rampActive THEN
    baseMasterRefRPM := instFB_Gen_SRamp.Y;

    // Automatically reset ramp flag when the ramp output reaches the target
    IF ABS(instFB_Gen_SRamp.Y - rampTargetRPM) <= 0.05 THEN
        rampActive := FALSE; // Ramp complete
    END_IF;

ELSE
    // No ramping required — direct assignment
    baseMasterRefRPM := rampTargetRPM;
END_IF;


(*
IF enableTorqueControl AND NOT enableTorqueControlOld THEN
	
	torqueSetpoint := torqueFeedback;
	
END_IF

enableTorqueControlOld := enableTorqueControl;
*)

IF NOT enableTorqueControl THEN
	
	instCTRL_PID_Group1TorqueTrim.LL := 0;
	instCTRL_PID_Group1TorqueTrim.LH := 0;
	
ELSE
	
	instCTRL_PID_Group1TorqueTrim.LL := torqueDifLimitLim;
	instCTRL_PID_Group1TorqueTrim.LH := torqueDifLimitMax;
	
END_IF



    instCTRL_PID_Group1TorqueTrim(
        ACT := torqueFeedback,
        SET := torqueSetpoint,
        MAN := FALSE,
        M_I := 0.0,
        RST := FALSE,
        KP  := torqueCtrlKp,
        TN  := torqueCtrlTn,
        TV  := torqueCtrlTv,
		SUP := 0.2,
        Y   => speedOffsetPID
    );

//--------------------------------------------------------------
// Operator offset (TUNE2 control)
//--------------------------------------------------------------
instTUNE2_GroupSpeedDiff(
    SET     := FALSE,
    SU      := groupSpeedDifInc,
    SD      := groupSpeedDifDec,
    RST     := FALSE,
    SS      := 0.01,
    FS      := 0.01,
    LIMIT_L := groupSpeedDifLimLow,
    LIMIT_H := groupSpeedDifLimHigh,
    Y       => groupSpeedOffset);

	
speedDif := groupSpeedOffset;
	
groupDeltaRatioAll  := 1.0 + ((speedOffsetPID + groupSpeedOffset) * 0.01);


//--------------------------------------------------------------
// Apply offsets + calculate all drive RPM references
//--------------------------------------------------------------
speedRefRPM := baseMasterRefRPM * groupDeltaRatioAll;


//--------------------------------------------------------------
// Convert RPM → MPM (surface speeds)
//--------------------------------------------------------------
group1MasterSpeedMPM := speedRefRPM * diameter * PI / 1000.0;


//--------------------------------------------------------------
// Suggest downstream handoff (group2 master surface speed)
//--------------------------------------------------------------
nextGroupSpeedRefMPM := group1MasterSpeedMPM;


//====================================================================
// ═══ PRIVATE METHOD — CALCULATE DIAMETER RATIOS ════════════════════
//====================================================================
METHOD PRIVATE _CalculateGearRatios
VAR_INPUT
END_VAR
;
END_METHOD

METHOD PRIVATE _Scale : REAL
VAR_INPUT
    X    : REAL;
    I_LO : REAL;
    I_HI : REAL;
    O_LO : REAL;
    O_HI : REAL;
END_VAR
IF I_LO = I_HI THEN
	_Scale := O_LO;
ELSE
	_Scale := (O_HI - O_LO) / (I_HI - I_LO) * (LIMIT(I_LO, X, I_HI) - I_LO) + O_LO;
END_IF;
END_METHOD

END_FUNCTION_BLOCK

// ---- Function Blocks/PaperMachine/DriveControl/FB_FormingBoardControl_V3.TcPOU
FUNCTION_BLOCK FB_FormingBoardControl_V3

VAR_INPUT

    //────────────────────────────────────────────
    // GROUP / INTERLOCKS
    //────────────────────────────────────────────
    startGroup              : BOOL; // Start command (pulse) / Comando de partida (pulso)
    stopGroup               : BOOL; // Stop command (level) / Comando de parada (nível)
    fastStopGroup               : BOOL; // Stop command (level) / Comando de parada (nível)
	groupReset              : BOOL; // Fault reset / Reset de falhas do grupo
	
    //────────────────────────────────────────────
    // AUXILIARY MOTORS — INDICATORS & COMMANDS
    //────────────────────────────────────────────
    grouSpeedDifIncCmd      : BOOL; // Lamp: offset increasing / Lâmpada: aumento de offset
    grouSpeedDifDecCmd      : BOOL; // Lamp: offset decreasing / Lâmpada: redução de offset
	
    //────────────────────────────────────────────
    // SPEED ADJUSTMENTS / OFFSET TUNING
    //────────────────────────────────────────────
    groupRecoverSpeedCmd    : BOOL; // Recover speed while TRUE / Recuperar velocidade enquanto TRUE
    //────────────────────────────────────────────
    // DRIVE STATUS INPUTS — FORMING BOARD ROLLS
    //────────────────────────────────────────────
    tractionRollReady       : BOOL; // MASTER ready / Pronto (mestre)
    suctionRollReady        : BOOL; // SLAVE ready / Pronto (seguidor)
	paperPresenceSensor : BOOL;

    //────────────────────────────────────────────
    // SPEED SETPOINTS / MODE
    //────────────────────────────────────────────
    groupAutoSpeedMPM       : REAL;       // Auto mode speed [m/min]
    groupManualSpeedMPM     : REAL := 50.0; // Manual mode speed
    groupSpeedAutoMan       : BOOL;       // 0=Manual, 1=Auto

    //────────────────────────────────────────────
    // SPEED & TORQUE FEEDBACKS
    //────────────────────────────────────────────
    tractionRollSpeedFeedback     : REAL; // MASTER speed feedback
    tractionRollTorqueFeedback    : REAL; // MASTER torque feedback
    suctionRollSpeedFeedback      : REAL; // SLAVE speed feedback
    suctionRollTorqueFeedback     : REAL; // SLAVE torque feedback

    //────────────────────────────────────────────
    // WIRE/FELT EDGE / RUNNING SAFETY SENSORS
    //────────────────────────────────────────────
    formingBoardWireOverrunSensorOperatorSide : BOOL; // Operator side / Lado operador
    formingBoardWireOverrunSensorDriveSide    : BOOL; // Drive side / Lado comando

    machineConfig : PaperMachine_TypeHmiConfig;

END_VAR



VAR_OUTPUT

    //────────────────────────────────────────────
    // STATE / DIAGNOSTICS
    //────────────────────────────────────────────
    deviceState                 : STRING; // Current state string / Estado atual em texto
    statusCode                  : INT;    // 0=Idle, 1=Starting, 2=Running, 3=Fault
    groupFault                  : BOOL;   // TRUE if any group fault active / Falha geral do grupo

    //────────────────────────────────────────────
    // SPEED REFERENCES (TO DRIVES) AND DISPLAY
    //────────────────────────────────────────────
    tractionRollSpeedSetpointRPM : REAL; // MASTER speed reference [rpm]
    suctionRollSpeedSetpointRPM  : REAL; // SLAVE speed reference [rpm]

    tractionRollSpeedFeedbackRPM : REAL; // MASTER speed feedback [rpm]
    suctionRollSpeedFeedbackRPM  : REAL; // SLAVE speed feedback [rpm]

    tractionRollSpeedFeedbackMPM : REAL; // MASTER speed feedback [m/min]
    suctionRollSpeedFeedbackMPM  : REAL; // SLAVE speed feedback [m/min]

    tractionRollTorqueFeedbackPct : REAL; // MASTER torque feedback [%]
    suctionRollTorqueFeedbackPct  : REAL; // SLAVE torque feedback [%]

    nextGroupSpeedRefMPM        : REAL; // Next group speed [m/min]

    //────────────────────────────────────────────
    // TORQUE REFERENCES / LIMITS (SLAVE)
    //────────────────────────────────────────────
    suctionRollTorqueRefPct     : REAL; // Torque setpoint for SLAVE [%]

    //────────────────────────────────────────────
    // DRIVE COMMANDS (ENABLE / RESET)
    //────────────────────────────────────────────
    tractionRollDriveEnable     : BOOL; // Enable MASTER drive
    tractionRollDriveReset      : BOOL; // Reset MASTER drive fault
    suctionRollDriveEnable      : BOOL; // Enable SLAVE drive
    suctionRollDriveReset       : BOOL; // Reset SLAVE drive fault

    //────────────────────────────────────────────
    // STATUS CODES (PER DRIVE)
    //────────────────────────────────────────────


    //────────────────────────────────────────────
    // HMI ALARMS STRUCTURE
    //────────────────────────────────────────────
    hmiAlarms                   : PaperMachine_TypeHmiAlarms;

END_VAR



VAR
    instFB_GroupDriveControl_V1       : FB_GroupDriveControl_V1;
    instFB_GroupSpeedControl_V1       : FB_GroupSpeedControl_V1;
	instFB_FormingBoardSpeedControl	: FB_FormingBoardSpeedControl;
    instFB_GroupDisplayFilters_V1     : FB_GroupDisplayFilters_V1;
    instFB_GroupTorqueTrimControl_V1  : FB_GroupTorqueTrimControl_V1;
	
	instFB_GroupTorqueTrimControl_V2  : FB_GroupTorqueTrimControl_V2;

	speedDif: REAL;
	speedDifError: BOOL;
	instTONWireOverRunTrip: TON;
END_VAR

VAR PERSISTENT
END_VAR

// ─────────────────────────────────────────────────────────────────────────────
// MAIN CALL SEQUENCE
// ─────────────────────────────────────────────────────────────────────────────

_GroupControl();          // 1) State machine: edges, enables, stop modes
_StateDisplay();
_SpeedDifferenceCheck();  // 4) Speed difference monitor & trip
_auxiliaryControls();

_alarmsDisplay();

METHOD _alarmsDisplay
VAR_INPUT
END_VAR
(*
//==============================================================
// FAULT EVALUATION — PER CONDITION (flags only; no global set)
//==============================================================

//----------------------------
// PRESS SECTION DRIVES
//----------------------------
hmiAlarms.pressSectionFirstPressFaultAlarm  := firstPressVfdFaultFeedback;
hmiAlarms.pressSectionSecondPressFaultAlarm := secondPressVfdFaultFeedback;

//----------------------------
// PRESS SECTION AUXILIARIES
//----------------------------
hmiAlarms.pressSectionUpperFeltStretcherFaultAlarm := upperFelt1StretcherFault;
hmiAlarms.pressSectionLowerFeltStretcherFaultAlarm := lowerFeltStretcherFault;
hmiAlarms.pressSectionUpperInfeedRollFaultAlarm    := upperInfeedRollFault;
hmiAlarms.pressSectionLowerInfeedRollFaultAlarm    := lowerInfeedRollFault;


//==============================================================
// PRESS SECTION — FELT EDGE OVERRUN ALARMS (DIRECT SENSORS)
//==============================================================

hmiAlarms.pressSectionUpperFelt1OverrunOperatorSideAlarm := pressSectionUpperFelt1OverrunSensorOperatorSide;
hmiAlarms.pressSectionUpperFelt1OverrunDriveSideAlarm    := pressSectionUpperFelt1OverrunSensorDriveSide;

hmiAlarms.pressSectionUpperFelt2OverrunOperatorSideAlarm := pressSectionUpperFelt2OverrunSensorOperatorSide;
hmiAlarms.pressSectionUpperFelt2OverrunDriveSideAlarm    := pressSectionUpperFelt2OverrunSensorDriveSide;

hmiAlarms.pressSectionLowerFeltOverrunOperatorSideAlarm := pressSectionLowerFeltOverrunSensorOperatorSide;
hmiAlarms.pressSectionLowerFeltOverrunDriveSideAlarm    := pressSectionLowerFeltOverrunSensorDriveSide;


//----------------------------
// PRESS SECTION GROUP FAULT STATUS
//----------------------------
groupFault :=
    hmiAlarms.pressSectionFirstPressFaultAlarm 
	OR hmiAlarms.pressSectionSecondPressFaultAlarm 
	OR hmiAlarms.pressFelt1OverrunOperatorSideAlarm
	OR hmiAlarms.pressFelt1OverrunDriveSideAlarm
	OR hmiAlarms.pressFelt2OverrunOperatorSideAlarm
	OR hmiAlarms.pressFelt2OverrunDriveSideAlarm
	OR hmiAlarms.pressFelt3OverrunOperatorSideAlarm
	OR hmiAlarms.pressFelt3OverrunDriveSideAlarm;


*)
//==============================================================
// FAULT EVALUATION — PER CONDITION (flags only; no global set)
//==============================================================

//----------------------------
// PRESS SECTION DRIVES
//----------------------------
//hmiAlarms.pressSectionFirstPressFaultAlarm  := firstPressVfdFaultFeedback;
//hmiAlarms.pressSectionSecondPressFaultAlarm := secondPressVfdFaultFeedback;

//----------------------------
// PRESS SECTION AUXILIARIES
//----------------------------
END_METHOD

METHOD _auxiliaryControls
VAR_INPUT
END_VAR
END_METHOD

METHOD _GroupControl
VAR_INPUT
END_VAR


(*
    formingBoardTorquePIDCtrlKp                   : REAL := 2.0;
    formingBoardTorquePIDCtrlTn                   : REAL := 8.0;
    formingBoardTorquePIDCtrlTv                   : REAL := 0.0;
    formingBoardTorqueLimit                   : REAL := 100.0;
	
*)
VAR
	suctionRollTorqueRefPct_: REAL;
END_VAR
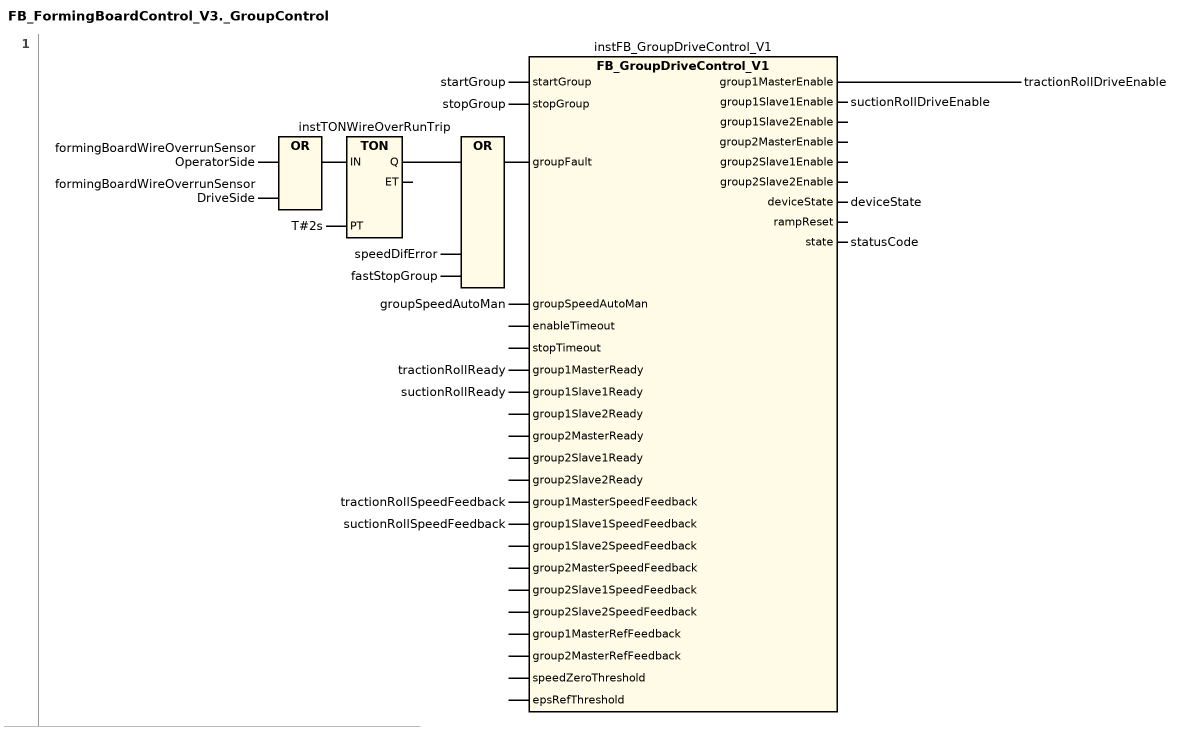
// NETWORK 1
instTONWireOverRunTrip(IN := formingBoardWireOverrunSensorOperatorSide OR formingBoardWireOverrunSensorDriveSide, PT := T#2s); // TON
instFB_GroupDriveControl_V1(
    startGroup := startGroup,
    stopGroup := stopGroup,
    groupFault := instTONWireOverRunTrip.Q OR speedDifError OR fastStopGroup,
    groupSpeedAutoMan := groupSpeedAutoMan,
    group1MasterReady := tractionRollReady,
    group1Slave1Ready := suctionRollReady,
    group1MasterSpeedFeedback := tractionRollSpeedFeedback,
    group1Slave1SpeedFeedback := suctionRollSpeedFeedback,
    group1Slave1Enable => suctionRollDriveEnable,
    deviceState => deviceState,
    state => statusCode); // FB_GroupDriveControl_V1
tractionRollDriveEnable := instFB_GroupDriveControl_V1.group1MasterEnable;

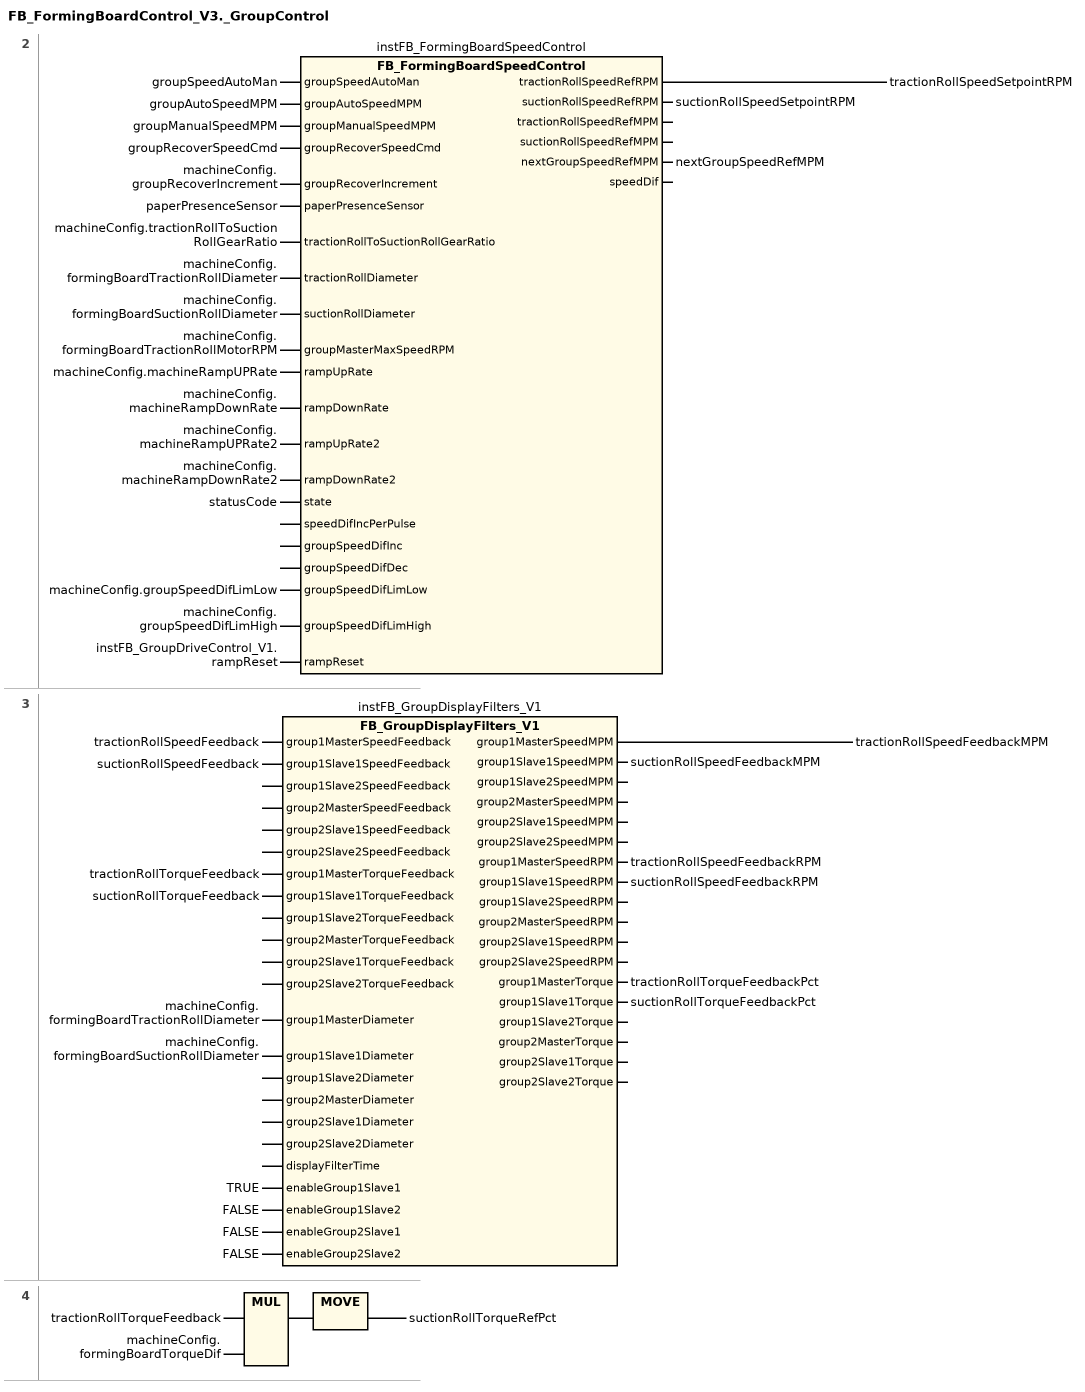
// NETWORK 2
instFB_FormingBoardSpeedControl(
    groupSpeedAutoMan := groupSpeedAutoMan,
    groupAutoSpeedMPM := groupAutoSpeedMPM,
    groupManualSpeedMPM := groupManualSpeedMPM,
    groupRecoverSpeedCmd := groupRecoverSpeedCmd,
    groupRecoverIncrement := machineConfig.groupRecoverIncrement,
    paperPresenceSensor := paperPresenceSensor,
    tractionRollToSuctionRollGearRatio := machineConfig.tractionRollToSuctionRollGearRatio,
    tractionRollDiameter := machineConfig.formingBoardTractionRollDiameter,
    suctionRollDiameter := machineConfig.formingBoardSuctionRollDiameter,
    groupMasterMaxSpeedRPM := machineConfig.formingBoardTractionRollMotorRPM,
    rampUpRate := machineConfig.machineRampUPRate,
    rampDownRate := machineConfig.machineRampDownRate,
    rampUpRate2 := machineConfig.machineRampUPRate2,
    rampDownRate2 := machineConfig.machineRampDownRate2,
    state := statusCode,
    groupSpeedDifLimLow := machineConfig.groupSpeedDifLimLow,
    groupSpeedDifLimHigh := machineConfig.groupSpeedDifLimHigh,
    rampReset := instFB_GroupDriveControl_V1.rampReset,
    suctionRollSpeedRefRPM => suctionRollSpeedSetpointRPM,
    nextGroupSpeedRefMPM => nextGroupSpeedRefMPM); // FB_FormingBoardSpeedControl
tractionRollSpeedSetpointRPM := instFB_FormingBoardSpeedControl.tractionRollSpeedRefRPM;

// NETWORK 3
instFB_GroupDisplayFilters_V1(
    group1MasterSpeedFeedback := tractionRollSpeedFeedback,
    group1Slave1SpeedFeedback := suctionRollSpeedFeedback,
    group1MasterTorqueFeedback := tractionRollTorqueFeedback,
    group1Slave1TorqueFeedback := suctionRollTorqueFeedback,
    group1MasterDiameter := machineConfig.formingBoardTractionRollDiameter,
    group1Slave1Diameter := machineConfig.formingBoardSuctionRollDiameter,
    enableGroup1Slave1 := TRUE,
    enableGroup1Slave2 := FALSE,
    enableGroup2Slave1 := FALSE,
    enableGroup2Slave2 := FALSE,
    group1Slave1SpeedMPM => suctionRollSpeedFeedbackMPM,
    group1MasterSpeedRPM => tractionRollSpeedFeedbackRPM,
    group1Slave1SpeedRPM => suctionRollSpeedFeedbackRPM,
    group1MasterTorque => tractionRollTorqueFeedbackPct,
    group1Slave1Torque => suctionRollTorqueFeedbackPct); // FB_GroupDisplayFilters_V1
tractionRollSpeedFeedbackMPM := instFB_GroupDisplayFilters_V1.group1MasterSpeedMPM;

// NETWORK 4
suctionRollTorqueRefPct := tractionRollTorqueFeedback * machineConfig.formingBoardTorqueDif;
END_METHOD

METHOD PRIVATE _Scale : REAL
VAR_INPUT
    X    : REAL;
    I_LO : REAL;
    I_HI : REAL;
    O_LO : REAL;
    O_HI : REAL;
END_VAR
IF I_LO = I_HI THEN
	_Scale := O_LO;
ELSE
	_Scale := (O_HI - O_LO) / (I_HI - I_LO) * (LIMIT(I_LO, X, I_HI) - I_LO) + O_LO;
END_IF;
END_METHOD

// ============================== Methods ==============================
// Intra-section speed supervision for Press Section (firstPress ↔ secondPress)
METHOD _SpeedDifferenceCheck
(*

    tractionRollSpeedFeedbackMPM : REAL; // MASTER speed feedback [m/min]
    suctionRollSpeedFeedbackMPM  : REAL; // SLAVE speed feedback [m/min]

*)


speedDif := ABS(tractionRollSpeedFeedbackMPM - suctionRollSpeedFeedbackMPM);


IF speedDif > 50 THEN
	
	speedDifError := TRUE;
	
	ELSE
		
	speedDifError := FALSE;
	
END_IF
END_METHOD

METHOD _StateDisplay
VAR_INPUT
END_VAR

// ──────────────────────────────────────────────────────────────────────────────
// _StateDisplay — Press Section (firstPress = Master, secondPress = Slave)
// Maps the internal machine "state" to a compact HMI status code and derives
// per-drive motor status codes from VFD signals.
//
// statusCode / firstPressStatusCode / secondPressStatusCode legend:
//   0 = Idle, 1 = Starting, 2 = Running, 3 = Fault
//
// Machine "state" groups:
//   0 = IDLE, 1 = ENABLE, 2 = WAIT_EN, 3 = RAMP_EN, 4 = RUN, 5 = STOPPING, 10 = FAULT
// Priority rule (for motors): Fault > Running > Starting > Idle
// ──────────────────────────────────────────────────────────────────────────────
VAR CONSTANT
    STATUS_IDLE     : INT := 0;
    STATUS_STARTING : INT := 1;
    STATUS_RUNNING  : INT := 2;
    STATUS_FAULT    : INT := 3;
END_VAR
END_METHOD

END_FUNCTION_BLOCK

// ---- Function Blocks/PaperMachine/FB_FormingBoardSpeedControl.TcPOU
FUNCTION_BLOCK FB_FormingBoardSpeedControl
VAR_INPUT
    //==============================================================
    // ─────────────── MODE SELECTION / REFERENCES ───────────────
    //==============================================================
    groupSpeedAutoMan          : BOOL;  // TRUE = Auto, FALSE = Manual
    groupAutoSpeedMPM          : REAL;  // Auto speed reference [m/min]
    groupManualSpeedMPM        : REAL;  // Manual speed reference [m/min]
    groupRecoverSpeedCmd       : BOOL;  // Recover (temporary speed bump)
    groupRecoverIncrement      : REAL;  // Recover increment [m/min]
//    interGroupGearRatio        : REAL;  // Inter-group ratio (next section sync)
	paperPresenceSensor				: BOOL;

    tractionRollToSuctionRollGearRatio  : REAL := 0.915;

    //==============================================================
    // ─────────────── DIAMETERS (mm) ───────────────
    //==============================================================
    tractionRollDiameter       : REAL;  // Diameter of group 1 master
    suctionRollDiameter       : REAL;  // Diameter of group 1 slave 1


    //==============================================================
    // ─────────────── CONFIGURATION / LIMITS ───────────────
    //==============================================================
    groupMasterMaxSpeedRPM     : REAL;  // Max allowed master RPM
    rampUpRate					: REAL := 0.1;  // Ramp slow acceleration [RPM/s]
    rampDownRate				: REAL := 0.1;  // Ramp slow acceleration [RPM/s]
	
    rampUpRate2					: REAL := 0.1;  // Ramp fast acceleration [RPM/s]
    rampDownRate2				: REAL := 0.1;  // Ramp fast acceleration [RPM/s]	
	
    state                      : INT;   // Machine state (5 = STOPPING)

	speedDifIncPerPulse		: REAL := 0.05;
	
    groupSpeedDifInc           : BOOL;  // Increment group speed offset
    groupSpeedDifDec           : BOOL;  // Decrement group speed offset
    groupSpeedDifLimLow        : REAL;  // Min offset [%]
    groupSpeedDifLimHigh       : REAL;  // Max offset [%]


    rampReset                  : BOOL;  // Reset ramp command
	
END_VAR


VAR_OUTPUT
    //==============================================================
    // ─────────────── FINAL DRIVE SPEEDS (RPM) ───────────────
    //==============================================================
    tractionRollSpeedRefRPM    : REAL; //Master speed
    suctionRollSpeedRefRPM    : REAL; // Slave speed

    //==============================================================
    // ─────────────── SURFACE SPEEDS (MPM) ───────────────
    //==============================================================
    tractionRollSpeedRefMPM       : REAL;
    suctionRollSpeedRefMPM       : REAL;


    //==============================================================
    // ─────────────── HANDOFF TO NEXT GROUP ───────────────
    //==============================================================
    nextGroupSpeedRefMPM       : REAL;
	speedDif					: REAL;
	
	
	
END_VAR


VAR
    //==============================================================
    // ─────────────── INTERNAL CALCULATION VARIABLES ───────────────
    //==============================================================
    masterMaxSpeedMPM          : REAL;
    baseCmdSpeedMPM            : REAL;
    cmdSpeedMPM                : REAL;
    targetRPM                  : REAL;
    rampTargetRPM              : REAL;
    baseMasterRefRPM           : REAL;
    groupSpeedOffset           : REAL;
    groupDeltaRatioAll         : REAL;
    upperLowerBiasRatio        : REAL;
    useRamp                    : BOOL;
    epsDiameter                : REAL := 0.001;

    // Gear ratios (set externally or calculated elsewhere)


    // Function blocks
    instFB_Gen_SRamp           : FB_Gen_SRamp;
    instFB_SpeedDif_SRamp           : FB_Gen_SRamp;

	rampActive: BOOL;
END_VAR


VAR PERSISTENT
	
    instTUNE2_GroupSpeedDiff   : TUNE2;

END_VAR

//==============================================================
// IMPLEMENTATION
//==============================================================

//====================================================================
// ═══ CALL METHOD TO CALCULATE DIAMETER RATIOS ═════════════════════
//====================================================================
_CalculateGearRatios();

//--------------------------------------------------------------
// Calculate master max surface speed [m/min]
//--------------------------------------------------------------
masterMaxSpeedMPM := groupMasterMaxSpeedRPM * (PI * tractionRollDiameter) / 1000.0;


//--------------------------------------------------------------
// Determine base speed source (auto/manual) + Recover bump
//--------------------------------------------------------------
IF groupSpeedAutoMan THEN
    baseCmdSpeedMPM := groupAutoSpeedMPM;
ELSE
    baseCmdSpeedMPM := groupManualSpeedMPM;
END_IF;

IF groupRecoverSpeedCmd THEN
    cmdSpeedMPM := baseCmdSpeedMPM + groupRecoverIncrement;
ELSE
    cmdSpeedMPM := baseCmdSpeedMPM;
END_IF;


//--------------------------------------------------------------
// Convert MPM → target RPM for the master
//--------------------------------------------------------------
targetRPM := _Scale(
    X    := cmdSpeedMPM,
    I_LO := 0.0,
    I_HI := masterMaxSpeedMPM,
    O_LO := 0.0,
    O_HI := groupMasterMaxSpeedRPM);


//--------------------------------------------------------------
// Ramp handling
//--------------------------------------------------------------
IF state = 5 OR state = 0 THEN
    // STOPPING — force ramp down to zero speed
    rampTargetRPM := 0.0;

ELSIF state = 10 THEN
    // FAULT — clear ramp immediately to ensure no residual motion
    rampTargetRPM := 0.0;
//    rampReset     := TRUE;

ELSE
    // Normal operation — ramp follows target speed
    rampTargetRPM := targetRPM;
//    rampReset     := FALSE;
END_IF;

// Detect when a new target speed change requires ramping
IF NOT rampActive AND ABS(rampTargetRPM - baseMasterRefRPM) >= 0.05 THEN
   rampActive := TRUE; // Rising edge — ramp request detected
 
END_IF;



IF 	paperPresenceSensor THEN
	//slow	
	instFB_Gen_SRamp.A_UP := MAX(0.0, rampUpRate);
	instFB_Gen_SRamp.A_DN := -MAX(0.0, rampDownRate);

ELSE
	//fast
	instFB_Gen_SRamp.A_UP := MAX(0.0, rampUpRate2);
	instFB_Gen_SRamp.A_DN := -MAX(0.0, rampDownRate2);

END_IF


// Ramp function block execution
instFB_Gen_SRamp(
    X          := rampTargetRPM,
//    A_UP       := MAX(0.0, rampUpRate),
//    A_DN       := -MAX(0.0, rampDownRate),
    VU_MAX     := 1000.0,
    VD_MAX     := -1000.0,
    LIMIT_HIGH := groupMasterMaxSpeedRPM,
    RST        := rampReset);

// If ramping, update the baseMasterRefRPM from ramp output
IF rampActive THEN
    baseMasterRefRPM := instFB_Gen_SRamp.Y;

    // Automatically reset ramp flag when the ramp output reaches the target
    IF ABS(instFB_Gen_SRamp.Y - rampTargetRPM) <= 0.05 THEN
        rampActive := FALSE; // Ramp complete
    END_IF;

ELSE
    // No ramping required — direct assignment
    baseMasterRefRPM := rampTargetRPM;
END_IF;


//--------------------------------------------------------------
// Operator offset (TUNE2 control)
//--------------------------------------------------------------
instTUNE2_GroupSpeedDiff(
    SET     := FALSE,
    SU      := groupSpeedDifInc,
    SD      := groupSpeedDifDec,
    RST     := FALSE,
    SS      := speedDifIncPerPulse,
    FS      := speedDifIncPerPulse,
    LIMIT_L := groupSpeedDifLimLow,
    LIMIT_H := groupSpeedDifLimHigh);
//    Y       => groupSpeedOffset);


// Ramp function block execution
instFB_SpeedDif_SRamp(
    X          := instTUNE2_GroupSpeedDiff.Y,
    A_UP       := MAX(0.0, 0.01),
    A_DN       := -MAX(0.0, 0.01),
    VU_MAX     := 1000.0,
    VD_MAX     := -1000.0,
    LIMIT_HIGH := groupSpeedDifLimHigh,
	LIMIT_LOW := groupSpeedDifLimLow,
    RST        := FALSE,
	Y => groupSpeedOffset);

	
speedDif := groupSpeedOffset;
	
groupDeltaRatioAll  := 1.0 + (groupSpeedOffset * 0.01);


//--------------------------------------------------------------
// Apply offsets + calculate all drive RPM references
//--------------------------------------------------------------
tractionRollSpeedRefRPM := baseMasterRefRPM * groupDeltaRatioAll;
suctionRollSpeedRefRPM := tractionRollSpeedRefRPM * tractionRollToSuctionRollGearRatio;


//--------------------------------------------------------------
// Convert RPM → MPM (surface speeds)
//--------------------------------------------------------------
tractionRollSpeedRefMPM := tractionRollSpeedRefRPM * tractionRollDiameter * PI / 1000.0;
suctionRollSpeedRefMPM := (suctionRollSpeedRefRPM * suctionRollDiameter * PI / 1000.0);



//--------------------------------------------------------------
// Suggest downstream handoff (group2 master surface speed)
//--------------------------------------------------------------
nextGroupSpeedRefMPM := tractionRollSpeedRefMPM;


//====================================================================
// ═══ PRIVATE METHOD — CALCULATE DIAMETER RATIOS ════════════════════
//====================================================================
METHOD PRIVATE _CalculateGearRatios
VAR_INPUT
END_VAR
END_METHOD

METHOD PRIVATE _Scale : REAL
VAR_INPUT
    X    : REAL;
    I_LO : REAL;
    I_HI : REAL;
    O_LO : REAL;
    O_HI : REAL;
END_VAR
IF I_LO = I_HI THEN
	_Scale := O_LO;
ELSE
	_Scale := (O_HI - O_LO) / (I_HI - I_LO) * (LIMIT(I_LO, X, I_HI) - I_LO) + O_LO;
END_IF;
END_METHOD

END_FUNCTION_BLOCK

// ---- Function Blocks/PaperMachine/Auxiliary/FB_SimpleMotorStart_V3.TcPOU
FUNCTION_BLOCK FB_SimpleMotorStart_V3
VAR_INPUT
    // ───────── Commands & interlocks ─────────
    startCommand                 : BOOL;   // Pulse to toggle run (Pulso para alternar execução)
    stopCommand                  : BOOL;   // Pulse to force stop (Pulso para forçar parada
	runtimeMeterResetCmd		: BOOL;
	
    motorStarterOK             : BOOL := TRUE;   // Softstarter healthy/ready (Softstarter ok/pronto)
    safetyOK                   	 : BOOL	:= TRUE;   // External interlock 1 (Intertravamento 1)
	
    interlock1                   : BOOL := TRUE;   // External interlock 2 (Intertravamento 2)
    interlock2                   : BOOL := TRUE;   // External interlock 3 (Intertravamento 3)
    interlock3                   : BOOL := TRUE;   // External interlock 4 (Intertravamento 4)

    // ───────── Motor current proof ─────────
    motorCurrentFeedback         : REAL;   // Measured motor current

END_VAR

VAR_OUTPUT
	
    faultActive                  : BOOL;       // Latched fault
	lineContactor                : BOOL;       // CMD line/bypass contactor
    deviceState                  : STRING(80); // Human-readable state
    statusCode                   : INT;        // 0=Idle, 1=Running, 2=Fault
    motorCurrentFiltered         : REAL;       // Filtered motor current for HMI/logic
	runtimeMeter				 : DINT;
	
END_VAR

VAR
    // ───────── State & edges ─────────
    step                         : INT;    // State machine step
    startCommandOld              : BOOL;
    stopCommandOld               : BOOL;
    rStart                       : BOOL;
    rStop                        : BOOL;

    // ───────── Latch ─────────
    runLatch                     : BOOL;   // Latched run request (start toggles, stop clears)

    // ───────── Timers ─────────
    tonStartDelay                : TON;    // Ramp-up timer

    // ───────── Helpers ─────────
    allInterlocksOK              : BOOL;
    proofCurrent                 : REAL;

    // ───────── OSCAT PT1 instance used by _InputFilter ─────────
    // Replace FT_PT1T with the correct type name from your OSCAT lib if different.
    instsFT_PT1TInputFilter      : FT_PT1;

END_VAR

// ============================ Edges, interlocks, defaults ============================
rStart := startCommand AND NOT startCommandOld;
rStop  := stopCommand  AND NOT stopCommandOld;
startCommandOld := startCommand;
stopCommandOld  := stopCommand;

allInterlocksOK := safetyOK AND interlock1 AND interlock2 AND interlock3;

// Start TOGGLES run latch; Stop forces stop
IF rStart THEN
    runLatch := NOT runLatch;  // Toggle / Alterna start-stop
END_IF;

IF rStop THEN
    runLatch := FALSE;         // Stop sempre desliga
END_IF;

// Default textual state
deviceState := 'Idle (Parado)';

// =============================== Fault reset =======================================
// Limpa falha somente quando não há pedido de partida e stop não está mantido
IF NOT runLatch AND NOT stopCommand THEN
    faultActive := FALSE;
END_IF;

// ============================= Interlocks & health checks ===========================
// Se pedir para rodar sem intertravamento ou softstarter OK -> entra em falha
IF runLatch AND NOT allInterlocksOK THEN
    faultActive := TRUE;
    deviceState := 'Fault: interlock open (Falha: intertrav. aberto)';
END_IF;

IF runLatch AND NOT motorStarterOK THEN
    faultActive := TRUE;
    deviceState := 'Fault: softstarter not OK (Falha: softstarter NOK)';
END_IF;

// Se falha ativa, garante tudo parado e volta pro passo 0
IF faultActive THEN
    lineContactor := FALSE;
    step := 0;
END_IF;

// ============================= Stop handling (immediate) ===========================
// Stop (pulso ou nível) força parada imediata
IF rStop OR stopCommand THEN
    lineContactor := FALSE;
    tonStartDelay(IN := FALSE);
    runLatch := FALSE;       // garante que o latch desligue
    step := 0;
END_IF;

// ================================= State machine ===================================
// Máquina de estados simples: 0 = Idle, 10 = Starting delay, 50 = Running
CASE step OF

    // ---------------------------------------------------------
    // 0: IDLE
    // ---------------------------------------------------------
    0:
        lineContactor := FALSE;
        tonStartDelay(IN := FALSE);
        deviceState := 'Idle (Parado)';

        // Condições para iniciar partida
        IF runLatch AND NOT faultActive AND motorStarterOK AND allInterlocksOK AND NOT stopCommand THEN
            // Inicia tempo de partida (ajuste o PT conforme desejado)
            tonStartDelay(IN := TRUE, PT := T#1S);
            deviceState := 'Starting (Partida - softstarter)';
            step := 10;
        END_IF;


    // ---------------------------------------------------------
    // 10: STARTING DELAY (SOFTSTARTER)
    // ---------------------------------------------------------
    10:
        deviceState := 'Starting (Partida - softstarter)';
        tonStartDelay(IN := TRUE, PT := T#3S);

        // Abort start se perder condição
        IF NOT runLatch OR stopCommand OR faultActive OR NOT allInterlocksOK OR NOT motorStarterOK THEN
            tonStartDelay(IN := FALSE);
            lineContactor := FALSE;
            step := 0;

        ELSIF tonStartDelay.Q THEN
            // Tempo de partida concluído -> liga contator de linha
            tonStartDelay(IN := FALSE);
            lineContactor := TRUE;
            step := 50;
        END_IF;


    // ---------------------------------------------------------
    // 50: RUNNING ON LINE
    // ---------------------------------------------------------
    50:
        lineContactor := TRUE;
        deviceState := 'Running on line (Operando em linha)';

        // Sai do RUN se o latch for desligado ou se der stop
        IF NOT runLatch OR stopCommand THEN
            lineContactor := FALSE;
            step := 0;
        END_IF;


    // ---------------------------------------------------------
    // Fallback (qualquer outro valor de step)
    // ---------------------------------------------------------
    ELSE
        lineContactor := FALSE;
        tonStartDelay(IN := FALSE);
        deviceState := 'Idle (Parado)';
        step := 0;
END_CASE;


// =============================== Status code =======================================
// 0 = Idle/Off
// 1 = Running
// 2 = Fault
IF faultActive THEN
    statusCode := 2;             // Fault
ELSIF lineContactor THEN
    statusCode := 1;             // Running
ELSE
    statusCode := 0;             // Idle / Off
END_IF;

// ============================================================================
// METHOD: _InputFilter
// OSCAT PT1 filter for PV, with enable/disable and bumpless behavior.
// When disabled, the filter tracks input quickly (tiny T) to avoid bumps.
// ============================================================================
METHOD PRIVATE _InputFilter
VAR_INPUT
    enableFilter   : BOOL;  // TRUE=apply PT1, FALSE=bypass
    rawValue       : REAL;  // Input value to be filtered
    filterTime     : TIME;  // PT1 time constant
    filterGainK    : REAL;  // PT1 gain, typically 1.0
END_VAR
VAR_OUTPUT
    filteredValue  : REAL;  // Filtered (or bypassed) value
END_VAR
VAR
    kUse           : REAL;
    tUse           : TIME;
    yPT1           : REAL;
END_VAR


IF enableFilter THEN
    kUse := filterGainK;
    tUse := filterTime;
ELSE
    // Track input closely for bumpless re-enable
    kUse := 1.0;
    tUse := T#10ms;
END_IF;

instsFT_PT1TInputFilter(
    in  := rawValue,
    T   := tUse,
    K   := kUse,
    out => yPT1
);

// Output selection
IF enableFilter THEN
    filteredValue := yPT1;
ELSE
    filteredValue := rawValue;
END_IF;
END_METHOD

END_FUNCTION_BLOCK

// ---- Function Blocks/PaperMachine/FB_AlarmControl.TcPOU
FUNCTION_BLOCK FB_AlarmControl
VAR_INPUT
	

	reset									: BOOL;
	
	formingBoardSafetyAlarm			: BOOL;
	pressSectionSafetyAlarm			: BOOL;
	dryingSectionSafetyAlarm		: BOOL;
	winderSectionSafetyAlarm		: BOOL;
	
	
   // ─────────────── FORMING BOARD ROLLS ───────────────
    formingBoardSuctionRollFaultAlarm         : BOOL;  // Suction roll fault / trip
    formingBoardSuctionRollCoolingFaultAlarm  : BOOL;  // Suction roll forced cooling fault
    formingBoardTractionRollFaultAlarm        : BOOL;  // Traction roll fault / trip
    formingBoardTractionRollCoolingFaultAlarm : BOOL;  // Traction roll forced cooling fault

    formingBoardRollDriveFaultAlarm           : BOOL;  // Roll up/down motor fault
    formingBoardStretchDriveFaultAlarm        : BOOL;  // Stretch motor fault

    // ── WIRE EDGE / RUNNING SAFETY SENSORS ─────────────────────────────────────
    formingBoardWireOverrunOperatorSideAlarm  : BOOL;  // Wire overrun detected on operator side (sensor active)
    formingBoardWireOverrunDriveSideAlarm     : BOOL;  // Wire overrun detected on drive side (sensor active)

    // ─────────────── PRESS SECTION DRIVES ───────────────
    pressSectionFirstPressFaultAlarm          : BOOL;  // First press (master) fault / trip
    pressSectionFirstPressCoolingFaultAlarm   : BOOL;  // First press forced cooling fault
    pressSectionSecondPressFaultAlarm         : BOOL;  // Second press (slave) fault / trip
    pressSectionSecondPressCoolingFaultAlarm  : BOOL;  // Second press forced cooling fault

    // ─────────────── PRESS SECTION — AUXILIARY MOTORS ───────────────
    pressSectionUpperFeltStretcherFaultAlarm  : BOOL;  // Upper felt stretcher motor fault / trip
    pressSectionLowerFeltStretcherFaultAlarm  : BOOL;  // Lower felt stretcher motor fault / trip
    pressSectionUpperInfeedRollFaultAlarm     : BOOL;  // Upper infeed roll motor fault / trip
    pressSectionLowerInfeedRollFaultAlarm     : BOOL;  // Lower infeed roll motor fault / trip

    // ── FELT EDGE / RUNNING SAFETY SENSORS ─────────────────────────────────────
    pressSectionUpperFelt1OverrunOperatorSideAlarm : BOOL;  // Felt 1 overrun detected on operator side (sensor active)
    pressSectionUpperFelt1OverrunDriveSideAlarm    : BOOL;  // Felt 1 overrun detected on drive side (sensor active)
    pressSectionUpperFelt2OverrunOperatorSideAlarm : BOOL;  // Felt 2 overrun detected on operator side (sensor active)
    pressSectionUpperFelt2OverrunDriveSideAlarm    : BOOL;  // Felt 2 overrun detected on drive side (sensor active)
    pressSectionLowerFeltOverrunOperatorSideAlarm  : BOOL;  // Felt 3 overrun detected on operator side (sensor active)
    pressSectionLowerFeltOverrunDriveSideAlarm     : BOOL;  // Felt 3 overrun detected on drive side (sensor active)

    // ─────────────── PRESS SECTION — GROUP FAULT ───────────────
    pressSectionGroupFaultAlarm               : BOOL;  // Global press section group fault / interlock active

    // ─────────────── DRYING SECTION — GROUP 1 ───────────────
    dryingSectionGroup1UpperMasterFaultAlarm         : BOOL;  // G1 Upper Master fault / trip
    dryingSectionGroup1UpperMasterCoolingFaultAlarm  : BOOL;  // G1 Upper Master forced cooling fault
    dryingSectionGroup1UpperSlave1FaultAlarm         : BOOL;  // G1 Upper Slave1 fault / trip
    dryingSectionGroup1UpperSlave1CoolingFaultAlarm  : BOOL;  // G1 Upper Slave1 forced cooling fault
    dryingSectionGroup1UpperSlave2FaultAlarm         : BOOL;  // G1 Upper Slave2 fault / trip
    dryingSectionGroup1UpperSlave2CoolingFaultAlarm  : BOOL;  // G1 Upper Slave2 forced cooling fault

    dryingSectionGroup1LowerMasterFaultAlarm         : BOOL;  // G1 Lower Master fault / trip
    dryingSectionGroup1LowerMasterCoolingFaultAlarm  : BOOL;  // G1 Lower Master forced cooling fault
    dryingSectionGroup1LowerSlave1FaultAlarm         : BOOL;  // G1 Lower Slave1 fault / trip
    dryingSectionGroup1LowerSlave1CoolingFaultAlarm  : BOOL;  // G1 Lower Slave1 forced cooling fault
    dryingSectionGroup1LowerSlave2FaultAlarm         : BOOL;  // G1 Lower Slave2 fault / trip
    dryingSectionGroup1LowerSlave2CoolingFaultAlarm  : BOOL;  // G1 Lower Slave2 forced cooling fault

    // ── FABRIC OVERRUN PROTECTION — GROUP 1 ───────────────────────────────────
    upperDryingSectionGroup1FabricOverrunOperatorSideAlarm : BOOL;  // Fabric overrun detected on operator side (sensor active)
    upperDryingSectionGroup1FabricOverrunDriveSideAlarm    : BOOL;  // Fabric overrun detected on drive side (sensor active)
    lowerDryingSectionGroup1FabricOverrunOperatorSideAlarm : BOOL;  // Fabric overrun detected on operator side (sensor active)
    lowerDryingSectionGroup1FabricOverrunDriveSideAlarm    : BOOL;  // Fabric overrun detected on drive side (sensor active)

    // ───────── DRYING SECTION — FABRIC STRETCHER — GROUP 1 ─────────
    upperDryingSectionGroup1FabricStretcherMotorFaultAlarm : BOOL;  // Upper fabric stretcher motor fault (G1)
    lowerDryingSectionGroup1FabricStretcherMotorFaultAlarm : BOOL;  // Lower fabric stretcher motor fault (G1)

    // ───────── DRYING SECTION — AUXILIARIES — GROUP 1 ─────────
    dryingSectionGroup1PickUpRollPosFaultAlarm       : BOOL;  // EN: G1 pick-up roll positioner fault / PT: Falha do posicionador do rolo pick-up G1
    dryingSectionGroup1BabyDryerScraperOscFaultAlarm : BOOL;  // EN: G1 babydryer scraper oscillator fault / PT: Falha do oscilador da raspa do babydryer G1
    dryingSectionGroup1UpperScraperOscFaultAlarm     : BOOL;  // EN: G1 upper group scraper oscillator fault / PT: Falha do oscilador da raspa do grupo superior G1
    dryingSectionGroup1LowerScraperOscFaultAlarm     : BOOL;  // EN: G1 lower group scraper oscillator fault / PT: Falha do oscilador da raspa do grupo inferior G1
    dryingSectionGroup1PaperBreakAlarm     : BOOL;  // EN: G1 lower group scraper oscillator fault / PT: Falha do oscilador da raspa do grupo inferior G1

    // ─────────────── DRYING SECTION — GROUP 2 ───────────────
    dryingSectionGroup2UpperMasterFaultAlarm         : BOOL;  // G2 Upper Master fault / trip
    dryingSectionGroup2UpperMasterCoolingFaultAlarm  : BOOL;  // G2 Upper Master forced cooling fault
    dryingSectionGroup2UpperSlave1FaultAlarm         : BOOL;  // G2 Upper Slave1 fault / trip
    dryingSectionGroup2UpperSlave1CoolingFaultAlarm  : BOOL;  // G2 Upper Slave1 forced cooling fault
    dryingSectionGroup2UpperSlave2FaultAlarm         : BOOL;  // G2 Upper Slave2 fault / trip
    dryingSectionGroup2UpperSlave2CoolingFaultAlarm  : BOOL;  // G2 Upper Slave2 forced cooling fault

    dryingSectionGroup2LowerMasterFaultAlarm         : BOOL;  // G2 Lower Master fault / trip
    dryingSectionGroup2LowerMasterCoolingFaultAlarm  : BOOL;  // G2 Lower Master forced cooling fault
    dryingSectionGroup2LowerSlave1FaultAlarm         : BOOL;  // G2 Lower Slave1 fault / trip
    dryingSectionGroup2LowerSlave1CoolingFaultAlarm  : BOOL;  // G2 Lower Slave1 forced cooling fault
    dryingSectionGroup2LowerSlave2FaultAlarm         : BOOL;  // G2 Lower Slave2 fault / trip
    dryingSectionGroup2LowerSlave2CoolingFaultAlarm  : BOOL;  // G2 Lower Slave2 forced cooling fault

    // ── FABRIC OVERRUN PROTECTION — GROUP 2 ───────────────────────────────────
    upperDryingSectionGroup2FabricOverrunOperatorSideAlarm : BOOL;  // Fabric overrun detected on operator side (sensor active)
    upperDryingSectionGroup2FabricOverrunDriveSideAlarm    : BOOL;  // Fabric overrun detected on drive side (sensor active)
    lowerDryingSectionGroup2FabricOverrunOperatorSideAlarm : BOOL;  // Fabric overrun detected on operator side (sensor active)
    lowerDryingSectionGroup2FabricOverrunDriveSideAlarm    : BOOL;  // Fabric overrun detected on drive side (sensor active)

    // ───────── DRYING SECTION — FABRIC STRETCHER — GROUP 2 ─────────
    upperDryingSectionGroup2FabricStretcherMotorFaultAlarm : BOOL;  // Upper fabric stretcher motor fault (G2)
    lowerDryingSectionGroup2FabricStretcherMotorFaultAlarm : BOOL;  // Lower fabric stretcher motor fault (G2)

    // ───────── DRYING SECTION — AUXILIARIES — GROUP 2 ─────────
    dryingSectionGroup2PickUpRollPosFaultAlarm       : BOOL;  // EN: G2 pick-up roll positioner fault / PT: Falha do posicionador do rolo pick-up G2
    dryingSectionGroup2BabyDryerScraperOscFaultAlarm : BOOL;  // EN: G2 babydryer scraper oscillator fault / PT: Falha do oscilador da raspa do babydryer G2
    dryingSectionGroup2UpperScraperOscFaultAlarm     : BOOL;  // EN: G2 upper group scraper oscillator fault / PT: Falha do oscilador da raspa do grupo superior G2
    dryingSectionGroup2LowerScraperOscFaultAlarm     : BOOL;  // EN: G2 lower group scraper oscillator fault / PT: Falha do oscilador da raspa do grupo inferior G2
    dryingSectionGroup2PaperBreakAlarm     : BOOL;  // EN: G1 lower group scraper oscillator fault / PT: Falha do oscilador da raspa do grupo inferior G1

    // ─────────────── DRYING SECTION — GROUP 3 ───────────────
    dryingSectionGroup3UpperMasterFaultAlarm         : BOOL;  // G3 Upper Master fault / trip
    dryingSectionGroup3UpperMasterCoolingFaultAlarm  : BOOL;  // G3 Upper Master forced cooling fault
    dryingSectionGroup3UpperSlave1FaultAlarm         : BOOL;  // G3 Upper Slave1 fault / trip
    dryingSectionGroup3UpperSlave1CoolingFaultAlarm  : BOOL;  // G3 Upper Slave1 forced cooling fault
    dryingSectionGroup3UpperSlave2FaultAlarm         : BOOL;  // G3 Upper Slave2 fault / trip
    dryingSectionGroup3UpperSlave2CoolingFaultAlarm  : BOOL;  // G3 Upper Slave2 forced cooling fault

    dryingSectionGroup3LowerMasterFaultAlarm         : BOOL;  // G3 Lower Master fault / trip
    dryingSectionGroup3LowerMasterCoolingFaultAlarm  : BOOL;  // G3 Lower Master forced cooling fault
    dryingSectionGroup3LowerSlave1FaultAlarm         : BOOL;  // G3 Lower Slave1 fault / trip
    dryingSectionGroup3LowerSlave1CoolingFaultAlarm  : BOOL;  // G3 Lower Slave1 forced cooling fault
    dryingSectionGroup3LowerSlave2FaultAlarm         : BOOL;  // G3 Lower Slave2 fault / trip
    dryingSectionGroup3LowerSlave2CoolingFaultAlarm  : BOOL;  // G3 Lower Slave2 forced cooling fault

    // ── FABRIC OVERRUN PROTECTION — GROUP 3 ───────────────────────────────────
    upperDryingSectionGroup3FabricOverrunOperatorSideAlarm : BOOL;  // Fabric overrun detected on operator side (sensor active)
    upperDryingSectionGroup3FabricOverrunDriveSideAlarm    : BOOL;  // Fabric overrun detected on drive side (sensor active)
    lowerDryingSectionGroup3FabricOverrunOperatorSideAlarm : BOOL;  // Fabric overrun detected on operator side (sensor active)
    lowerDryingSectionGroup3FabricOverrunDriveSideAlarm    : BOOL;  // Fabric overrun detected on drive side (sensor active)

    // ───────── DRYING SECTION — FABRIC STRETCHER — GROUP 3 ─────────
    upperDryingSectionGroup3FabricStretcherMotorFaultAlarm : BOOL;  // Upper fabric stretcher motor fault (G3)
    lowerDryingSectionGroup3FabricStretcherMotorFaultAlarm : BOOL;  // Lower fabric stretcher motor fault (G3)

    // ───────── DRYING SECTION — AUXILIARIES — GROUP 3 ─────────
    dryingSectionGroup3PickUpRollPosFaultAlarm       : BOOL;  // EN: G3 pick-up roll positioner fault / PT: Falha do posicionador do rolo pick-up G3
    dryingSectionGroup3BabyDryerScraperOscFaultAlarm : BOOL;  // EN: G3 babydryer scraper oscillator fault / PT: Falha do oscilador da raspa do babydryer G3
    dryingSectionGroup3UpperScraperOscFaultAlarm     : BOOL;  // EN: G3 upper group scraper oscillator fault / PT: Falha do oscilador da raspa do grupo superior G3
    dryingSectionGroup3LowerScraperOscFaultAlarm     : BOOL;  // EN: G3 lower group scraper oscillator fault / PT: Falha do oscilador da raspa do grupo inferior G3
    dryingSectionGroup3PaperBreakAlarm     : BOOL;  // EN: G1 lower group scraper oscillator fault / PT: Falha do oscilador da raspa do grupo inferior G1

    // ─────────────── CENTRIFUGAL PRESSURE SCREEN ───────────────
    cpsUnitFaultAlarm                        : BOOL;  // Screen unit fault / trip

    // ─────────────── COUCH PIT PUMP & MIXER ───────────────
    couchPitPumpFaultAlarm                   : BOOL;  // Couch pit pump fault / trip

    // ─────────────── WIRE PIT PUMP ───────────────
    wirePitPumpFaultAlarm                    : BOOL;  // Wire pit pump fault / trip

    // ─────────────── STOCK PUMP ───────────────
    stockPumpFaultAlarm                      : BOOL;  // Stock pump fault / trip

    // ─────────────── MIXING PUMP ───────────────
    mixingPumpFaultAlarm                     : BOOL;  // Mixing pump fault / trip

    // ─────────────── VACUUM PUMPS ───────────────
    vacuumPump1FaultAlarm                    : BOOL;  // Vacuum pump 1 fault / trip
    vacuumPump2FaultAlarm                    : BOOL;  // Vacuum pump 2 fault / trip

    // ─────────────── LOW VACUUM EXHAUST FAN ───────────────
    lowVacuumFanFaultAlarm                   : BOOL;  // Low vacuum exhaust fan fault / trip

    // ─────────────── LUBRIFICATION PUMPS ───────────────
    lubricationPump1FaultAlarm              : BOOL;  // Lubrication pump 1 fault / trip
    lubricationPump2FaultAlarm              : BOOL;  // Lubrication pump 2 fault / trip
    lubricationMinPressureFaultAlarm        : BOOL;  // Minimum pressure not reached / trip
    lubricationMaxPressureFaultAlarm        : BOOL;  // Overpressure in lubrication circuit / trip
	lubricationTankHighTemperatureAlarm 	: BOOL;
	lubricationCircuitHighTemperatureAlarm 	: BOOL;

END_VAR
VAR_OUTPUT
	
    alarmsDisplay    : PaperMachine_TypeHmiAlarms;
	alarmIndication	: BOOL;

END_VAR
VAR
	
    alarmsVariables    : PaperMachine_TypeHmiAlarms;

	resetOld: BOOL;
END_VAR

_00_Reset();
_01_FormingBoardAlarms();
_02_PressSectionAlarms();
_03_DryingSectionAlarms();
_04_WinderSectionAlarms();
_08_AlarmIndication();

METHOD _00_Reset
VAR_INPUT
END_VAR
IF reset AND NOT resetOld THEN
	
	//Copy values from a holder variable with zero value to reset
	alarmsDisplay := alarmsVariables;
	
END_IF
END_METHOD

METHOD _01_FormingBoardAlarms
VAR_INPUT
END_VAR
IF formingBoardSafetyAlarm THEN
	
	alarmsDisplay.formingBoardSafetyAlarm := TRUE;

END_IF

//────────────────────────────────────────────
// FORMING BOARD — ROLLS & DRIVES
//────────────────────────────────────────────
IF formingBoardSuctionRollFaultAlarm THEN
    alarmsDisplay.formingBoardSuctionRollFaultAlarm := TRUE;
END_IF

IF formingBoardSuctionRollCoolingFaultAlarm THEN
    alarmsDisplay.formingBoardSuctionRollCoolingFaultAlarm := TRUE;
END_IF

IF formingBoardTractionRollFaultAlarm THEN
    alarmsDisplay.formingBoardTractionRollFaultAlarm := TRUE;
END_IF

IF formingBoardTractionRollCoolingFaultAlarm THEN
    alarmsDisplay.formingBoardTractionRollCoolingFaultAlarm := TRUE;
END_IF

IF formingBoardRollDriveFaultAlarm THEN
    alarmsDisplay.formingBoardRollDriveFaultAlarm := TRUE;
END_IF

IF formingBoardStretchDriveFaultAlarm THEN
    alarmsDisplay.formingBoardStretchDriveFaultAlarm := TRUE;
END_IF


//────────────────────────────────────────────
// FORMING BOARD — WIRE EDGE / RUNNING SAFETY
//────────────────────────────────────────────
IF formingBoardWireOverrunOperatorSideAlarm THEN
    alarmsDisplay.formingBoardWireOverrunOperatorSideAlarm := TRUE;
END_IF

IF formingBoardWireOverrunDriveSideAlarm THEN
    alarmsDisplay.formingBoardWireOverrunDriveSideAlarm := TRUE;
END_IF
END_METHOD

METHOD _02_PressSectionAlarms
VAR_INPUT
END_VAR
//────────────────────────────────────────────
// PRESS SECTION — DRIVES
//────────────────────────────────────────────
IF pressSectionFirstPressFaultAlarm THEN
    alarmsDisplay.pressSectionFirstPressFaultAlarm := TRUE;
END_IF

IF pressSectionFirstPressCoolingFaultAlarm THEN
    alarmsDisplay.pressSectionFirstPressCoolingFaultAlarm := TRUE;
END_IF

IF pressSectionSecondPressFaultAlarm THEN
    alarmsDisplay.pressSectionSecondPressFaultAlarm := TRUE;
END_IF

IF pressSectionSecondPressCoolingFaultAlarm THEN
    alarmsDisplay.pressSectionSecondPressCoolingFaultAlarm := TRUE;
END_IF


//────────────────────────────────────────────
// PRESS SECTION — AUXILIARY MOTORS
//────────────────────────────────────────────
IF pressSectionUpperFeltStretcherFaultAlarm THEN
    alarmsDisplay.pressSectionUpperFeltStretcherFaultAlarm := TRUE;
END_IF

IF pressSectionLowerFeltStretcherFaultAlarm THEN
    alarmsDisplay.pressSectionLowerFeltStretcherFaultAlarm := TRUE;
END_IF

IF pressSectionUpperInfeedRollFaultAlarm THEN
    alarmsDisplay.pressSectionUpperInfeedRollFaultAlarm := TRUE;
END_IF

IF pressSectionLowerInfeedRollFaultAlarm THEN
    alarmsDisplay.pressSectionLowerInfeedRollFaultAlarm := TRUE;
END_IF


//────────────────────────────────────────────
// PRESS SECTION — FELT EDGE / RUNNING SAFETY
//────────────────────────────────────────────
IF pressSectionUpperFelt1OverrunOperatorSideAlarm THEN
    alarmsDisplay.pressSectionUpperFelt1OverrunOperatorSideAlarm := TRUE;
END_IF

IF pressSectionUpperFelt1OverrunDriveSideAlarm THEN
    alarmsDisplay.pressSectionUpperFelt1OverrunDriveSideAlarm := TRUE;
END_IF

IF pressSectionUpperFelt2OverrunOperatorSideAlarm THEN
    alarmsDisplay.pressSectionUpperFelt2OverrunOperatorSideAlarm := TRUE;
END_IF

IF pressSectionUpperFelt2OverrunDriveSideAlarm THEN
    alarmsDisplay.pressSectionUpperFelt2OverrunDriveSideAlarm := TRUE;
END_IF

